SYMBOL_TABLE
"DB_Message"	DB 2	UDT 2
"INS_ZERO_POINT_SYSTEM"	DB 15	FB 15	// Instanzbaustein Nullpunktspannsystem
"INS_CLAMPING_SYSTEM"	DB 17	FB 17	// Instanz-DB Spannsystem (hydraulisch, pneumatisch)
"INS_MESSAGE_OUT"	DB 100	FB 100	// Arbeitsdaten Alarm-/Meldungserfassung
"DB_CK_OP"	DB 101	UDT 101	// DB für Überwachung von Operanden
"DB_IN"	DB 111	DB 111	// Kommunikation - Eingänge
"DB_OUT"	DB 112	DB 112	// Kommunikation - Ausgänge
"ZERO_POINT_SYSTEM"	FB 15	FB 15	// Nullpunktspannsystem
"CLAMPING_SYSTEM"	FB 17	FB 17	// Spannsystem (hydraulisch, pneumatisch)
"AutoSusDoor"	FB 20	FB 20	// pneum.Rüstplatztüren
"MESSAGE_OUT"	FB 100	FB 100	// Ausgabe Alarm-/Betriebsmeldungen
"FlowMonitoring"	FC 10	FC 10	// Strömungsüberwachung
"HydraulicMonitoring"	FC 12	FC 12	// Überwachung Hydrauliksystem (Filter, ...)
"OperatingData"	FC 30	FC 30	// Betriebsdatenerfassung, Signalleuchte (-säule, Ampel)
"MonitoringFuse"	FC 33	FC 33	// Erfassung und Auswertung der Sicherungen
"MontioringCircuitBreaker"	FC 34	FC 34	// Erfassung und Auswertung der Leistungsschalter
"MonitoringMainDrive"	FC 35	FC 35
"ChipConveyor"	FC 42	FC 42
"COOLANT"	FC 50	FC 50	// Kühlmittel Druckerhöhung
"FUNCTIONS"	FC 90	FC 90	// allgemeine Funktionen
"CHANGE_BYTE"	FC 91	FC 91
"SIGNAL"	FC 92	FC 92	// allgemeine Signalverknüpfungen
"SELECT_TIME"	FC 93	FC 93	// aus MD (2Dekaden) 2 Zeitwerte (Time) erzeugen
"MachineType"	FC 94	FC 94	// Dekodierung des Maschinentyps und Optionen aus einem Maschinenparameter
"FC_CK2OP"	FC 101	FC 101	// Überwachung von 2 Operanden
"FC_CK1OP"	FC 102	FC 102	// Überwachung eines Operanden
"INPUT_MASTER"	FC 111	FC 111	// Eingänge von Mastersystem lesen
"OUTPUT_MASTER"	FC 112	FC 112	// Ausgänge an Mastersystem schreiben
"CallAutoSusDoor"	FC 120	FC 120
"INPUT_PERIPHERIE"	FC 121	FC 121	// Eingänge von Peripherie lesen
"OUTPUT_PERIPHERIE"	FC 122	FC 122	// Ausgänge an Peripherie schreiben
"M_LOW"	M 0.0	BOOL	// Merker mit Zustand Low  "FALSE"
"M_HIGH"	M 0.1	BOOL	// Merker mit Zustand High  "TRUE"
"m_expertenbit"	M 0.2	BOOL	// Expertenbit für Fehleranzeige
"M_STARTPULSE"	M 0.5	BOOL	// Startimpuls, wird nur einmalig, für einen Zyklus gesetzt.
"m_inbetriebnahme"	M 0.6	BOOL
"m_konstruktion"	M 0.7	BOOL
"M_TAKT_0.1SEC"	M 1.0	BOOL	// Taktmerker 0.1sec/10Hz
"M_TAKT_0.2SEC"	M 1.1	BOOL	// Taktmerker 0.2sec/5Hz
"M_TAKT_0.4SEC"	M 1.2	BOOL	// Taktmerker 0.4sec/2.5Hz
"M_TAKT_0.5SEC"	M 1.3	BOOL	// Taktmerker 0.5sec/2Hz
"M_TAKT_0.8SEC"	M 1.4	BOOL	// Taktmerker 0.8sec/1.25Hz
"M_TAKT_1.0SEC"	M 1.5	BOOL	// Taktmerker 1.0sec/1Hz
"M_TAKT_1.6SEC"	M 1.6	BOOL	// Taktmerker 1.6sec/0.625Hz
"M_TAKT_2.0SEC"	M 1.7	BOOL	// Taktmerker 2.0sec/0.5Hz
"M_MESSAGE"	M 50.0	BOOL	// Zwischenspeicher für Meldung "PW-Freigabe nicht möglich"
"M_Hyd_Filter_Alarm"	M 50.1	BOOL	// Zwischenspeicher für Hydraulik Filter Alarm
"M_Hyd_Füll_Warn"	M 50.2	BOOL	// Zwischenspeicher für Hydraulik Füllstand Warnung
"M_Hyd_Füll_Alarm"	M 50.3	BOOL	// Zwischenspeicher für Hydraulik Füllstand Alarm
"M_Hyd_Temp_Alarm"	M 50.4	BOOL	// Zwischenspeicher für Hydraulik Temperatur Alarm
"mTypeDMUxxP2"	M 60.1	BOOL	// (1) Maschinenbaureihe DMU xxP2
"mType1"	M 60.2	BOOL
"mType2"	M 60.3	BOOL
"mType3"	M 60.4	BOOL
"mTypeDMCxxU2"	M 60.5	BOOL	// (5) Maschinenbaureihe DMC xxU2
"mTypeDMCxxU2RS"	M 60.6	BOOL	// (6) Maschinenbaureihe DMC xxU2 mit Rundspeicher
"mTypeDMCxxU2WS"	M 60.7	BOOL	// (7) Maschinenbaureihe DMC xxU2 mit Werkstückspeicher (Fastems)
"mType4"	M 61.0	BOOL
"mType5"	M 61.1	BOOL
"mType6"	M 61.2	BOOL
"mType7"	M 61.3	BOOL
"mType8"	M 61.4	BOOL
"mType9"	M 61.5	BOOL
"mType10"	M 61.6	BOOL
"mType11"	M 61.7	BOOL
"mPalletClampingHead"	M 62.0	BOOL	// (256) Palettenausführung mit Spannköpfen/Spannkonen
"mTurnTable"	M 62.1	BOOL	// (512) Fräs-Drehtisch
"mOption2"	M 62.2	BOOL	// (1024)
"mOption3"	M 62.3	BOOL	// (2048)
"mOption4"	M 62.4	BOOL	// (4096)
"mOption5"	M 62.5	BOOL	// (8192)
"mOption6"	M 62.6	BOOL	// (16384)
"mOption7"	M 62.7	BOOL	// (32768)
"mOption8"	M 63.4	BOOL	// (16)
"mOption9"	M 63.5	BOOL	// (32)
"mOption10"	M 63.6	BOOL	// (64)
"mOption11"	M 63.7	BOOL	// (128)
"Flankenmerker_1"	M 80.0	BOOL	// Zwischenspeicher für Flankenauswertung 1
"Flankenmerker_2"	M 80.1	BOOL	// Zwischenspeicher für Flankenauswertung 2
"Flankenmerker_3"	M 80.2	BOOL	// Zwischenspeicher für Flankenauswertung 3
"Flankenmerker_4"	M 80.3	BOOL	// Zwischenspeicher für Flankenauswertung 4
"Flankenmerker_5"	M 80.4	BOOL	// Zwischenspeicher für Flankenauswertung 5
"Flankenmerker_6"	M 80.5	BOOL	// Zwischenspeicher für Flankenauswertung 5
"Flankenmerker_7"	M 80.6	BOOL	// Zwischenspeicher für Flankenauswertung 5
"Flankenmerker_8"	M 80.7	BOOL	// Zwischenspeicher für Flankenauswertung 5
"Hilfsmerker_1"	M 90.0	BOOL	// Zwischenspeicher 1
"Hilfsmerker_2"	M 90.1	BOOL	// Zwischenspeicher 2
"Hilfsmerker_3"	M 90.2	BOOL	// Zwischenspeicher 3
"Hilfsmerker_4"	M 90.3	BOOL	// Zwischenspeicher 4
"Hilfsmerker_5"	M 90.4	BOOL	// Zwischenspeicher 5
"Hilfsmerker_6"	M 90.5	BOOL	// Zwischenspeicher 6
"Hilfsmerker_7"	M 90.6	BOOL	// Zwischenspeicher 7
"Hilfsmerker_8"	M 90.7	BOOL	// Zwischenspeicher 8
"EpxCoolantFlowM7"	M 100.0	BOOL	// Durchflusswächter Kühlmittel2 (M7)
"EpxWireFlowSensorOkM7"	M 100.1	BOOL	// /Durchflusswächter HD Leitungsüberwachung
"EpxCoolantFlowM8"	M 100.2	BOOL	// Durchflusswächter Kühlmittel1 (M8)
"EpxWireFlowSensorOkM8"	M 100.3	BOOL	// /Durchflusswächter ND Leitungsüberwachung
"EPX_ZPS_RELEASE"	M 100.4	BOOL	// Nullpunktspannsystem lösen
"EPX_ZPS_LOCKED"	M 100.5	BOOL	// Nullpunktspannsystem gesperrt
"EPX_ZPS_PRESSURE_MIN1"	M 100.6	BOOL	// Nullpunktspannsystem Drucküberwachung_1 Minimaldruck (p~0) = gespannt
"EPX_ZPS_PRESSURE_MIN2"	M 100.7	BOOL	// Nullpunktspannsystem Drucküberwachung_2 Minimaldruck (p~0) = gespannt
"EPX_ZPS_PRESSURE_MAX1"	M 101.0	BOOL	// Nullpunktspannsystem Drucküberwachung_1 Maximaldruck (p=max) = gelöst
"EPX_ZPS_PRESSURE_MAX2"	M 101.1	BOOL	// Nullpunktspannsystem Drucküberwachung_2 Maximaldruck (p=max) = gelöst
"EPX_COOLANT_LIMIT_VALUE"	M 101.2	BOOL	// /Füllstandsüberwachung im Sammelbehälter
"EPX_LUBRICATION_LEVEL"	M 101.3	BOOL	// Füllstandsüberwachung Schmierstoffaggregat
"EPX_ZPS_MODE_AUTO"	M 101.4	BOOL	// Nullpunktspannsystem in Betriebsart Automatik = Ansteuerung durch ext. Einheit
"EPX_ZPS_INTERLOCK_MIN1"	M 101.5	BOOL	// Nullpunktspannsystem - Verriegelungskontrolle Druck ~0 (drucklos)
"EPX_ZPS_INTERLOCK_MAX1"	M 101.6	BOOL	// Nullpunktspannsystem - Verriegelungskontrolle Druck vorhanden (=verriegelt)
"EPX_ZPS_DISTANCE_P_MIN1"	M 101.7	BOOL	// Nullpunktspannsystem - Auflagenkontrolle Druck ~0 (drucklos)
"EPX_ZPS_DISTANCE_P_MAX1"	M 102.0	BOOL	// Nullpunktspannsystem - Auflagenkontrolle Druck erreicht (Präzision vorhanden)
"EPX_ALARM_QUIT"	M 102.1	BOOL	// Rücksetzen der Fehlermeldung (z.B. Akustik)
"EPX_EL-CABINETDOOR1_OPEN"	M 102.2	BOOL	// Schaltschranktür(-kombination)_1 der Werkzeugmaschine geöffnet
"EPX_EL-CABINETDOOR2_OPEN"	M 102.3	BOOL	// Schaltschranktür(-kombination)_2 der Werkzeugmaschine geöffnet
"EPX_EL-CABINETDOOR5_OPEN"	M 102.4	BOOL	// Schaltschranktür(-kombination)_1 der Kühlschmierstoffanlage geöffnet
"EPX_EL_CABINET_TEMP_1"	M 102.5	BOOL	// Uebertemperatur Schaltschrank Werkzeugmaschine
"EPX_EL_CABINET_TEMP_2"	M 102.6	BOOL	// Grenzwertmeldung Schaltschranktemperatur Werkzeugmaschine
"EPX_EL-CABINETDOOR3_OPEN"	M 102.7	BOOL	// Schaltschranktür(-kombination)_3 der Werkzeugmaschine geöffnet
"EPX_SO_APC_POS_180"	M 103.0	BOOL	// Palettenwechsler Stellung 180 Grad (Palette_2 im Arbeitsraum)
"EPX_SO_APC_POS_0"	M 103.1	BOOL	// Palettenwechsler Stellung 0 Grad (Palette_1 im Arbeitsraum)
"EPX_VCS_MODE_MIXED"	M 103.2	BOOL	// Anwahl Betriebsart <Vakuumsystem Mischbetrieb> aktiv
"EPX_VCS_MODE_VACUUM"	M 103.3	BOOL	// Anwahl Betriebsart <Vakuumsystem Vollwechsel> aktiv
"EPX_VCS_MODE_OFF"	M 103.4	BOOL	// Anwahl Betriebsart <Vakuumsystem Aus>
"EPX_VCS_READY_1"	M 103.5	BOOL	// Betriebsbereitmeldung Vakuumsystem (Arbeitsraum) z.B. Leistungssschalter, ...
"EPX_VCS_READY_2"	M 103.6	BOOL	// Betriebsbereitmeldung Vakuumsystem (Rüstplatz) z.B. Leistungssschalter, ...
"EPX_VCS_RELEASE_FIXTURE2"	M 103.7	BOOL	// Vakuumspannsystem am Rüstplatz lösen
"EPX_VCS_FIXTURE1_1_P=0"	M 104.0	BOOL	// Vakuumspannsystem im Arbeitsraum Drucklos (=gelöst)
"EPX_VCS_FIXTURE1_2_P=0"	M 104.1	BOOL	// Vakuumspannsystem im Arbeitsraum Drucklos (=gelöst)
"EPX_VCS_FIXTURE2_1_P=0"	M 104.2	BOOL	// Vakuumspannsystem am Rüstplatz Drucklos (=gelöst)
"EPX_VCS_FIXTURE1_1_P=MAX"	M 104.3	BOOL	// Vakuumspannsystem im Arbeitsraum gespannt (eingestellter Sollwert erreicht)
"EPX_VCS_FIXTURE2_1_P=MAX"	M 104.4	BOOL	// Vakuumspannsystem am Rüstplatz gespannt (eingestellter Sollwert erreicht)
"EpxHydrFilterAlarm1NC"	M 104.5	BOOL	// Filterverschmutzung Hydraulikfilter-Maschine (Alarm 100%)
"EpxHydrFilterWarning1NC"	M 104.6	BOOL	// Filterverschmutzung Hydraulikfilter-Maschine (Warnung 75%)
"EPX_EXH_NEG_READY1"	M 104.7	BOOL	// Auswertung Leistungsschalter des Nebelabscheiders_1/Absaugung_1
"EPX_EXH_ON1"	M 105.0	BOOL	// Überwachung Ansteuerung Nebelabscheider_1, Gerät ein
"EPX_MACHINE_ON_K1"	M 105.1	BOOL	// "Maschine Ein"-Signal an Kühlschmierstoffanlage (kein Not-Aus)
"EPX_WORKROOM_CLOSED_K1"	M 105.2	BOOL	// "Arbeitsraumtüren geschlossen"-Signal an Kühlschmierstoffanlage
"EPX_NEG_COO_MESSAGE"	M 105.3	BOOL	// Warnmeldung von Kühlschmierstoffanlage
"EPX_NEG_COO_ALARM"	M 105.4	BOOL	// Störung, Alarm von Kühlschmierstoffanlage
"EPX_COO_ACK_COOLANT2.2"	M 105.5	BOOL	// Rückmeldung wenn Druckstufe_2 von Kühlmittel_2 erreicht wurde (YD-Anlauf)
"EPX_COO_MAINVALVE_CLOSED"	M 105.6	BOOL	// Kühlschmierstoffzufuhr Haupt-/Zentralventil geschlossen
"EPX_COO_PRESSURE_P=MAX"	M 105.7	BOOL	// Kühlschmierstoffzufuhr Drucküberwachung
"EPX_COO_MAIN_FLOW"	M 106.0	BOOL	// Kühlschmierstoffzufuhr Durchflussüberwachung
"EPX_COO_LIMITVALUE_K5"	M 106.1	BOOL	// Grenzwertmeldung aus Sammelbehälter (SPF) z.B. von WHG-Sonde
"EPX_NEG_COO_FILTALARM2.2"	M 106.2	BOOL	// Filterverschmutzung Feinfilter Alarmmeldung für KSS-Zufuhr_2 (IKZ)-Druckstufe_2
"EPX_COO_FILTWARN2.2"	M 106.3	BOOL	// Filterverschmutzung Feinfilter Warnmeldung für KSS-Zufuhr_2 (IKZ) - Druckstufe_2
"EPX_VCS_RELEASE_FIXTURE1"	M 106.4	BOOL	// Vakuumspannsystem im Arbeitsraum lösen
"EPX_CS_OFF"	M 106.5	BOOL	// Spannsystem deaktiviert, Aus
"EPX_CS_MODE_AUTO"	M 106.6	BOOL	// Spannsystem in der Betriebsart "AUTOMATIK" (=externe Ansteuerung)
"EPX_CS_RELEASE1_1"	M 106.7	BOOL	// Anforderung Spannsystem lösen im Arbeitsraum (Spannkreis 1)
"EPX_CS_PRESSURE1_1MIN"	M 107.0	BOOL	// Spannsystem DruckÜW im Arbeitsraum (Spannkreis 1/Stufe 1 - Systemdruck Min)
"EPX_CS_PRESSURE1_1MAX"	M 107.1	BOOL	// Spannsystem DruckÜW im Arbeitsraum (Spannkreis 1/Stufe 1 - Systemdruck Max)
"EPX_CS_PRESSURE1_2MIN"	M 107.2	BOOL	// Spannsystem DruckÜW im Arbeitsraum (Spannkreis 1/Stufe 2 - Lösedruck Min)
"EPX_CS_PRESSURE1_2MAX"	M 107.3	BOOL	// Spannsystem DruckÜW im Arbeitsraum (Spannkreis 1/Stufe 2 - Lösedruck Max)
"EPX_CS_STROKE1_POS1"	M 107.4	BOOL	// Spannsystem Hubkontrolle im Arbeitsraum (Werkstück gelöst)
"EPX_CS_STROKE1_POS2"	M 107.5	BOOL	// Spannsystem Hubkontrolle im Arbeitsraum (Werkstück gespannt)
"EPX_CS_STROKE1_POS3"	M 107.6	BOOL	// Spannsystem Hubkontrolle im Arbeitsraum (gespannt ohne Werkstück)
"EPX_EXT_FIXTURE_EXIST"	M 107.7	BOOL	// Werkstück an Spannvorrichtung, Spannfutter (Signal von externer Einheit)
"EPX_EXT_RELEASE1"	M 108.0	BOOL	// Anforderung Spannsystem lösen im Arbeitsraum (Signal von externer Einheit)
"EPX_APC_DOOR_CLOSED"	M 108.1	BOOL	// Rüstplatztüren geschlossen (NICHT verriegelt)
"EPX_EXH_ON2"	M 108.2	BOOL	// Überwachung Ansteuerung Nebelabscheider_2, Gerät ein
"EPX_EXH_NEG_READY2"	M 108.3	BOOL	// Auswertung Leistungsschalter des Nebelabscheiders_2/Absaugung_2
"EPX_EXH_SELECT1"	M 108.4	BOOL	// Absaugung - Auswahl für Nebelabscheider_1
"EPX_EXH_SELECT2"	M 108.5	BOOL	// Absaugung - Auswahl für Nebelabscheider_2
"EPX_MCS_CLAMP1"	M 108.6	BOOL	// Magnetspannsystem_1 spannen
"EPX_MCS_RELEASE1"	M 108.7	BOOL	// Magnetspannsystem_1 lösen
"EPX_MCS_PARK_STATION1"	M 109.0	BOOL	// Magnetspannsystem_1 Magnetisierungsstecker am Ablageplatz (Parkstation)-Rpl
"EPX_MCS_LOCKED1"	M 109.1	BOOL	// Magnetspannsystem_1 Betriebsart gesperrt/deaktiviert
"EPX_HYD_FILTER_OK1"	M 109.2	BOOL	// Filter des Hydraulikaggregates-Maschine in Ordnung
"EPX_COO_ACK_COOLANT2.1"	M 109.3	BOOL	// Rückmeldung wenn Druckstufe_1 von Kühlmittel_2 erreicht wurde (YD-Anlauf)
"EPX_ZPS_RELEASE1_START"	M 109.4	BOOL	// Nullpunktspannsystem lösen - Startsignal, direkt vom Befehlsgerät
"EPX_SRT_SWIVELPOS=0"	M 109.5	BOOL	// Schwenkrundtisch - Schwenkachse steht in horizontaler Position (0 Grad)
"EPX_CS_FINALPOS0"	M 109.6	BOOL	// Spannvorrichtung - Endlage Position 0 erreicht
"EPX_CS_FINALPOS1"	M 109.7	BOOL	// Spannvorrichtung - Endlage Position 1 erreicht
"EPX_CS_NOT_FINALPOS0"	M 110.0	BOOL	// Spannvorrichtung - Endlage Position 0  NICHT erreicht/vorhanden
"EPX_CS_NOT_FINALPOS1"	M 110.1	BOOL	// Spannvorrichtung - Endlage Position 1  NICHT erreicht/vorhanden
"EPX_CS_PRESSURIZED_POS0"	M 110.2	BOOL	// Spannvorrichtung - Druck vorhanden für Bewegung auf Position 0
"EPX_CS_PRESSURIZED_POS1"	M 110.3	BOOL	// Spannvorrichtung - Druck vorhanden für Bewegung auf Position 1
"EPX_CS_ROTATECONTROL_ON"	M 110.4	BOOL	// Spannvorrichtung - Überwachung der Drehbewegung aktiviert
"EPX_COO_FLUSH1_P=SYST"	M 110.5	BOOL	// Drucküberwachung Kühlschmierstoffzufuhr Spänespülung(en) = Systemdruck
"EPX_COO_FLUSH1_P=MAX"	M 110.6	BOOL	// Drucküberwachung Kühlschmierstoffzufuhr Spänespülung(en) = maximaler Druck
"EPX_ZPS_ENABLE"	M 110.7	BOOL	// Nullpunktspannsystem gespannt oder nicht aktiviert (?HLS?)
"EPX_MMS_FILLUNIT_NIV_MIN"	M 111.0	BOOL	// MMS: Versorgungseinheit - Füllstand Minimum
"EPX_MMS_NIVEAU_MIN"	M 111.1	BOOL	// MMS: Füllstand Minimum
"EPX_MMS_NIVEAU_MAX"	M 111.2	BOOL	// MMS: Füllstand Maximum
"EPX_MMS_NIVEAU_WAR_MIN"	M 111.3	BOOL	// MMS: Füllstand Minimum - Vorwarnung
"EPX_SPINDLE_FEED_STOP"	M 111.4	BOOL	// Spindel- und Vorschub Halt (allgemein)
"EPX_VCS_FIXTURE_START1"	M 111.5	BOOL	// Vakuumsystem lösen (Startsignal)
"EPX_MCS_MODE_ON1"	M 111.6	BOOL	// Magnetspannsystem (Hauptschalter Ein)
"EPX_ZPS_CYL_LIFT"	M 111.7	BOOL	// Nullpunktspannsystem Abhebezylinder heben (ausfahren)
"EPX_ZPS_CYL_LOWER"	M 112.0	BOOL	// Nullpunktspannsystem Abhebezylinder senken (einfahren)
"EPX_ZPS_CYL_PRESS_MIN1"	M 112.1	BOOL	// Nullpunktspannsystem Abhebezylinder Heben Druck Minimum   (p~0) = eingefahren
"EPX_ZPS_CYL_PRESS_MIN2"	M 112.2	BOOL	// Nullpunktspannsystem Abhebezylinder Senken Druck Minimum   (p~0) = ausgefahren
"EPX_ZPS_CYL_PRESS_MAX1"	M 112.3	BOOL	// Nullpunktspannsystem Abhebezylinder Heben Druck Maximum   (p~max) = ausgefahren
"EPX_ZPS_CYL_PRESS_MAX2"	M 112.4	BOOL	// Nullpunktspannsystem Abhebezylinder Senken Druck Maximum   (p~max) = eingefahren
"EpxFunctionM86"	M 112.5	BOOL	// maschinenspezifische Funktion (M86)
"EpxFunctionM87"	M 112.6	BOOL	// maschinenspezifische Funktion (M87)
"EpxFunctionM88"	M 112.7	BOOL	// maschinenspezifische Funktion (M88)
"EpxFunctionM89"	M 113.0	BOOL	// maschinenspezifische Funktion (M89)
"EpxMcsParkshutterLocked"	M 113.1	BOOL	// Magnetspannsystem Parkstation Klappe geschlossen
"EpxMcsAntiSteckParks"	M 113.2	BOOL	// Magnetspannsystem Stecker nicht vorhanden
"EpxMcsParkstatEnable"	M 113.3	BOOL	// Magnetspannsystem Parkstation entriegelt
"EpxMcsPlugIn"	M 113.4	BOOL	// Magnetspannsystem Stecker in Magnetspannplatte
"EpxMcsOff"	M 113.5	BOOL	// Magnetspannsystem aus
"EpxMcsEnableRelease"	M 113.6	BOOL	// Magnetspannsystem Freigabe lösen
"EpxMcsMaleInParkstaion"	M 113.7	BOOL	// Magnetspannsystem Stecker in Parkstation
"EpxMcsAdhesivForceOk"	M 114.0	BOOL	// Magnetspannsystem eingestellte Haftkraftstufe erreicht
"EpxCooPwarnSupfineLevel"	M 114.1	BOOL	// Vorwarnung Füllstand Kühlschmierstoff im Feinbereich
"EpxCooEnergyCentrifugeOk"	M 114.2	BOOL	// Überwachung Leistungsschalter der Zentrifuge
"EpxCooCentrifugeReady"	M 114.3	BOOL	// Zentrifuge Betreibsbereit
"EpxCooCentrifugeRun"	M 114.4	BOOL	// Zentrifuge in Betrieb
"EpxCooPwarnCentrifugeQui"	M 114.5	BOOL	// Vorwarnung der Zentrifuge zurücksetzen
"EPX_ZPS_CS1_PRESSLES"	M 114.6	BOOL	// Abfrage des Spanndruckes der Spannhydraulik Kreis 1
"EPX_ZPS_CS2_PRESSLES"	M 114.7	BOOL	// Abfrage des Spanndruckes der Spannhydraulik Kreis 2
"EpxExhausterModeAuto"	M 115.0	BOOL	// Automatikbetrieb Absaugung Ölnebelabscheider
"EPX_SAMMELSTÖRUNG_1"	M 115.1	BOOL	// Meldung von externer Meldeeinrichtung
"EPX_SAMMELSTÖRUNG_2"	M 115.2	BOOL	// Meldung von externer Meldeeinrichtung
"EpxCooNoLimitCollBasin"	M 115.3	BOOL	// keine Grenzwertmeldung Sammelbehälter (WHG)
"EpxEmergStopMachineNC"	M 115.4	BOOL	// Kein Not-Aus an Werkzeugmaschine betätigt
"EpxEmergStopPanel"	M 115.5	BOOL	// Not-Aus Pilzdrucktaster an Bedienpult (Werkzeugmaschine) betätigt
"EpxEmergStopChipConv"	M 115.6	BOOL	// Not-Aus Pilzdrucktaster am Späneförderer betätigt
"EpxEmergStopSetUpStat"	M 115.7	BOOL	// Not-Aus Pilzdrucktaster am Rüstplatz (Palettenspeicher) betätigt
"EpxEmergStopToolInpStat"	M 116.0	BOOL	// Not-Aus Pilzdrucktaster an der Werkzeugeingabestation betätigt
"EpxLubricatPressureXaxis"	M 116.1	BOOL	// Drucküberwachung Schmierung Verteiler X-Achse Ok
"EpxLubricatPressureYaxis"	M 116.2	BOOL	// Drucküberwachung Schmierung Verteiler Y-Achse Ok
"EpxLubricatPressureZaxis"	M 116.3	BOOL	// Drucküberwachung Schmierung Verteiler Z-Achse Ok
"EpxFaultExtChipConveyNC"	M 116.4	BOOL	// LOW = Störung an externem (zentralen) Späneförderer
"EpxLimitValveCoolantNC"	M 116.5	BOOL	// LOW = maximaler Füllstand (Grenzwert) der Kühlschmierstoffanlage erreicht/übers.
"EpxMaintDoorToolInpStat"	M 116.6	BOOL	// Wartungstüre Werkzeugeingabestation offen
"EpxMaintDoorToolMag"	M 116.7	BOOL	// Wartungstüre Werkzeugmagazin offen
"EpxMaintDoorPalletStor"	M 117.0	BOOL	// Wartungstüre Palettenspeicher/-wechsler offen
"EpxLubTablePreExi"	M 117.1	BOOL	// NC-Rundtisch Schmierung Druck Vorhanden
"EpxEmergStopHaWhToolMag"	M 117.2	BOOL	// Not-Aus Pilzdrucktaster des Handrad vom Werkzeugmagazin betätigt
"EpxLubTableApsOk"	M 117.3	BOOL	// Schmierstoffpumpe Leistungsschalter Ok
"EpxLubXAxisPreExi1"	M 117.4	BOOL	// Drucküberwachung Schmierung Verteiler KUG X-Achse
"EpxLubYAxisPreExi1"	M 117.5	BOOL	// Drucküberwachung Schmierung Verteiler KUG Y-Achse
"EpxLubPcAxisPreExi"	M 117.6	BOOL	// Drucküberwachung Schmierung Verteiler Palettenspeichersystem (Palettenwechsler)
"EpxLubSstAxisPreExi"	M 117.7	BOOL	// Drucküberwachung Schmierung Verteiler Ruestplatz
"EpxFusePlugIndicPlate"	M 118.0	BOOL	// Überwachung Sicherungsautomat Steckdose Frontschild
"EpxFuseLubPump"	M 118.1	BOOL	// Überwachung Sicherungsautomat Schmierstoffpumpe
"EpxFuseAsi"	M 118.2	BOOL	// Überwachung Sicherungsautomat AS-i Netzteil
"EpxFuseFlowControl"	M 118.3	BOOL	// Überwachung Sicherungsautomat Durchflusswächter
"EpxFuseLightBulbs"	M 118.4	BOOL	// Überwachung Sicherungsautomat Leuchtmelder Kommandostation
"EpxFuseControlCircuit"	M 118.5	BOOL	// Überwachung Sicherungsautomat Steuerstromkreis
"EpxFuseCncControl"	M 118.6	BOOL	// Überwachung Sicherungsautomat CNC-Steuerung
"EpxFuseEmpStopConCircuit"	M 118.7	BOOL	// Überwachung Sicherungsautomat NOT-AUS Steuerstromkreis
"EpxFuseToolChanger"	M 119.0	BOOL	// Überwachung Sicherungsautomat Werkzeugwechsler
"EpxFuseDcControlVoltage"	M 119.1	BOOL	// Überwachung Sicherungsautomat DC-Steuerspannung
"EpxFusePalletChanger"	M 119.2	BOOL	// Überwachung Sicherungsautomat Palettenwechsler
"EpxFuseCoolantUnit"	M 119.3	BOOL	// Überwachung Sicherungsautomat Kühlmittelanlage
"EpxFusePcu50"	M 119.4	BOOL	// Überwachung Sicherungsautomat PCU 50
"EpxFuseScreen"	M 119.5	BOOL	// Überwachung Sicherungsautomat Bildschirm
"EpxFuseMachineIm151_4"	M 119.6	BOOL	// Überwachung Sicherungsautomat Maschine IM 151
"EpxFuseMachineOutp1Im151"	M 119.7	BOOL	// Überwachung Sicherungsautomat Ausgänge Maschine IM 151
"EpxFuseMachineOutp2Im151"	M 120.0	BOOL	// Überwachung Sicherungsautomat Ausgänge Maschine IM 151
"EpxFuseSpeedControl"	M 120.1	BOOL	// Überwachung Sicherungsautomat Drehzahl Überwachung
"EpxFusePowerPacTc"	M 120.2	BOOL	// Überwachung Sicherungsautomat Netzteil Werkzeugwechsler
"EpxFuseToolIdentificatio"	M 120.3	BOOL	// Überwachung Sicherungsautomat Werkzeugidentifikation
"EpxFuseToolCone"	M 120.4	BOOL	// Überwachung Sicherungsautomat Werkzeugkegel
"EpxFuseControCirPis"	M 120.5	BOOL	// Überwachung Sicherungsautomat Palettenspeichersystem
"EpxFuseBrakePs"	M 120.6	BOOL	// Überwachung Sicherungsautomat Palettenspeichersystem Bremse
"EpxFuseOperaDataRecord"	M 120.7	BOOL	// Überwachung Sicherungsautomat Betriebsdatenerfassung
"EpxFuseToolBrake"	M 121.0	BOOL	// Überwachung Sicherungsautomat Werkzeugbruchüberwachung
"EpxFuseMms"	M 121.1	BOOL	// Überwachung Sicherungsautomat Minimalmengenschmierung
"EpxFuseSlave8"	M 121.2	BOOL	// Überwachung Sicherungsautomat Tuning IM 151
"EpxFuseSlave8Output"	M 121.3	BOOL	// Überwachung Sicherungsautomat Tuning Ausgänge IM 151
"EpxFuseSlave8Input"	M 121.4	BOOL	// Überwachung Sicherungsautomat Tuning Eingänge IM 151
"EpxFuseCabinetLightning"	M 121.5	BOOL	// Überwachung Sicherungsautomat Schaltschrankbeleuchtung
"EpxCuFuseSensor"	M 121.6	BOOL	// Überwachung Sicherungsautomat Sensoren Kühlmittelanlage
"EpxCuFusePropValve1"	M 121.7	BOOL	// Überwachung Sicherungsautomat Proportionalventil 1 Kühlmittelanlage
"EpxCuFusePropValve2"	M 122.0	BOOL	// Überwachung Sicherungsautomat Proportionalventil 2 Kühlmittelanlage
"EpxCuApsCoolant1"	M 122.1	BOOL	// Überwachung Leistungsschalter Kühlmittel 1
"EpxCuApsFlushCleaTop"	M 122.2	BOOL	// Überwachung Leistungsschalter Spänespülung Dach
"EpxCuApsFlushGun"	M 122.3	BOOL	// Überwachung Leistungsschalter Spülpistole
"EpxCuApsFlushCleaCabDoor"	M 122.4	BOOL	// Überwachung Leistungsschalter Spänespülung Kabinentür
"EpxCuApsSuperfineRegion"	M 122.5	BOOL	// Überwachung Leistungsschalter Feinstbereich
"EpxCuApsTroughScraper"	M 122.6	BOOL	// Überwachung Leistungsschalter Kratzerförderer
"EpxCuMainSwitch"	M 122.7	BOOL	// Überwachung Hauptschalter Kühlmittelanlage
"EpxCuApsPump40bar"	M 123.0	BOOL	// Überwachung Leistungsschalter Hochdruckpumpe 40 bar
"EpxCuApsPump80bar"	M 123.1	BOOL	// Überwachung Leistungsschalter Hochdruckpumpe 80 bar
"EpxCuTempApsCompressor"	M 123.2	BOOL	// Überwachung Leistungsschalter Kompressor Kühlaggregat
"EpxCuTempApsFan"	M 123.3	BOOL	// Überwachung Leistungsschalter Lüfter Kühlaggregat
"EpxCuTempApsAgitator"	M 123.4	BOOL	// Überwachung Leistungsschalter Rührwerk Kühlaggregat
"EpxCuTempApsLiftingPump"	M 123.5	BOOL	// Überwachung Leistungsschalter Hebepumpe Kühlaggregat
"EpxCuTempApsHeating"	M 123.6	BOOL	// Überwachung Leistungsschalter Heizung Kühlaggregat
"EpxCuTempApsContrVoltage"	M 123.7	BOOL	// Überwachung Leistungsschalter Steuerspannung Kühlaggregat
"EpxApsCabinetLightning"	M 124.0	BOOL	// Überwachung Leistungsschalter Schaltschrankbeleuchtung
"EpxApsDcControlVoltage1"	M 124.1	BOOL	// Überwachung Leistungsschalter DC-Steuerspannung 1
"EpxApsDcControlVoltage2"	M 124.2	BOOL	// Überwachung Leistungsschalter DC-Steuerspannung 2
"EpxApsAcControlVoltage"	M 124.3	BOOL	// Überwachung Leistungsschalter AC-Steuerspannung
"EpxApsTemperature"	M 124.4	BOOL	// Überwachung Leistungsschalter Kuehl/Heizaggregat
"EpxApsPowerSupplyModule"	M 124.5	BOOL	// Überwachung Leistungsschalter AC-Versorgungsmodul
"EpxMcsParkStation2"	M 124.6	BOOL	// Magnetspannsystem_2 Magnetisierungsstecker am Ablageplatz (Parkstation)-Maschine
"EpxMcsReleased"	M 124.7	BOOL	// Magnetspannplatte gelöst
"EpxMcsChucked"	M 125.0	BOOL	// Magnetspannplatte gespannt
"EpxMcsMalfunction"	M 125.1	BOOL	// Magnetspannsystem Störung
"EpxFeedStop"	M 125.2	BOOL	// Vorschub Halt
"EpxFuseMachineIm151_7"	M 125.3	BOOL	// Überwachung Sicherungsautomat Maschine IM 151_7
"EpxFuseSpeedControlSst"	M 125.4	BOOL	// Überwachung Sicherungsautomat Drehzahl Überwachung Rüstplatz
"EpxFuseMeasuringSensor"	M 125.5	BOOL	// Überwachung Sicherungsautomat Messtaster
"EpxFuseWorkingAreaDoor"	M 125.6	BOOL	// Überwachung Sicherungsautomat Kabinentüre
"EpxTmsFuseBrake"	M 125.7	BOOL	// Überwachung Sicherungsautomat Bremse Regalmagazin
"EpxTmsFuseAcContrVoltage"	M 126.0	BOOL	// Überwachung Sicherungsautomat AC-Steuerspannung Regalmagazin
"EpxTmsFuseControlCircuit"	M 126.1	BOOL	// Überwachung Sicherungsautomat Steuerstromkreis Regalmagazin
"EpxTmsFuseControlPanel"	M 126.2	BOOL	// Überwachung Sicherungsautomat Werkzeugeingabestation Regalmagazin
"EpxTmsFuseOutput"	M 126.3	BOOL	// Überwachung Sicherungsautomat Ausgänge Regalmagazin
"EpxTmsFusePowerPac"	M 126.4	BOOL	// Überwachung Sicherungsautomat Netzteil Regalmagazin
"EpxTmsApsPower"	M 126.5	BOOL	// Überwachung Leistungschalter Netzeinspeisung Regalmagazin
"EpxLubTmsAxisPreExi"	M 126.6	BOOL	// Drucküberwachung Schmierung Verteiler Werkzeugmagazin
"EpxFuseFeedDrive"	M 126.7	BOOL	// Überwachund Sicherungsautomat Leistung Spindel
"EpxMaintDoorToolShelf"	M 127.0	BOOL	// Wartungstüre Werkzeugregal offen
"EpxApsAcControVoltageFan"	M 127.1	BOOL	// Überwachung Leistungsschalter Lüfter AC
"EpxApsAcCoolCabinet"	M 127.2	BOOL	// Überwachung Leistungsschalter Kühlaggregat Schaltschrank
"EpxApsPowerToolShelf"	M 127.3	BOOL	// Überwachung Leistungsschalter Werkzeugregal
"EpxApsFdFan"	M 127.4	BOOL	// Überwachung Leistungsschalter Lüfter FD
"EpsApsCoolingUnit"	M 127.5	BOOL	// Überwachung Leistungsschalter Kühlmittelanlage
"EpxTmsApsAcControlVoltag"	M 127.6	BOOL	// Überwachung Leistungsschalter Steuerspannung AC-Regalmagazin
"EpxTmsApsDrives"	M 127.7	BOOL	// Überwachung Leistungsschalter Antriebe Regalmagazin
"EpxHydFuellMaxOk"	M 128.0	BOOL	// Füllstand Hydraulik Maximum Ok
"EpxHydFuellMinOk"	M 128.1	BOOL	// Füllstand Hydraulik Minimum Ok
"EpxFuse230V"	M 128.2	BOOL	// Überwachung Sicherungsautomaten 230V
"EpxFuse24V"	M 128.3	BOOL	// Überwachung Sicherungsautomaten 24V
"EpxApsContPanelPlugSock"	M 128.4	BOOL	// Überwachung Leistungsschalter Steckdose Bedienpult
"EpxApsPcPlugSock"	M 128.5	BOOL	// Überwachung Leistungsschalter Steckdose Palettenwechsler-/speichersystem
"EpxSusDoorSystPressMax"	M 128.6	BOOL	// Ruestplatztürantreib Systemdruck vorhanden
"EpxCloseSusDoor"	M 128.7	BOOL	// Rüstplatztüre(n) schliessen (manuelle Bedienung)
"EpxOpenSusDoor"	M 129.0	BOOL	// Rüstplatztüre(n) öffnen (manuelle Bedienung)
"EpxRobotLock"	M 129.1	BOOL	// Betreibsart Werkstücklader gesperrt = manuelles Beladen
"EpxSafetyEdgeSusDoor"	M 129.2	BOOL	// Schaltleiste an Rüstplatztüren betätigt
"EpxSusDoorPressMonOpen"	M 129.3	BOOL	// Drucküberwachung Rüstplatztüren öffnen aktiv
"EpxSusDoorPressMonClose"	M 129.4	BOOL	// Drucküberwachung Rüstplatztüren schließen aktiv
"EpxSusDoorLeftOpen"	M 129.5	BOOL	// Rüstplatztüre links vollständig geöffnet
"EpxSusDoorRightOpen"	M 129.6	BOOL	// Rüstplatztüre rechts vollständig geöffnet
"EpxSusDoorClosed"	M 129.7	BOOL	// Rüstplatztüre(n) geschlossen
"EpxSusDoorClosedLocked"	M 130.0	BOOL	// Rüstplatztüre(n) geschlossen und verriegelt
"EpxPressMonitLubToolMag"	M 130.1	BOOL	// Drucküberwachung Schmierung Werkzeugmagazin
"EpxCircBrkMachineOutpNc"	M 130.2	BOOL	// Überwachung Leitungsschutzschalter Ausgänge IM151 (Maschine)
"EpxCircBrkCtlVoToolMagNc"	M 130.3	BOOL	// Überwachung Leitungsschutzschalter Steuerstromkreis Werkzeugmagazin
"EpxPowSwitchAddCoolng1Nc"	M 130.4	BOOL	// Überwachung Leitungsschutzschalter Kühlaggregat Zusatzschaltschrank (Einspeisung
"EpxApsWorkingAreaDoor"	M 130.5	BOOL	// Überwachung Leistungschutzschalter Kabinentüre
"EpxMachineOn"	M 130.6	BOOL	// Maschine ist eingeschaltet (kein Not-Aus)
"EpxProgramRun"	M 130.7	BOOL	// Programm läuft
"EpxLubDec1Bit_0"	M 131.0	BOOL	// Schmierimpuls Binär codiert Bit 0
"EpxLubDec1Bit_1"	M 131.1	BOOL	// Schmierimpuls Binär codiert Bit 1
"EpxLubDec1Bit_2"	M 131.2	BOOL	// Schmierimpuls Binär codiert Bit 2
"EpxLubDec1Bit_3"	M 131.3	BOOL	// Schmierimpuls Binär codiert Bit 3
"EpxLubDec1Bit_4"	M 131.4	BOOL	// Schmierimpuls Binär codiert Bit 4
"EpxLubDec1Bit_5"	M 131.5	BOOL	// Schmierimpuls Binär codiert Bit 5
"EpxLubDec1Bit_6"	M 131.6	BOOL	// Schmierimpuls Binär codiert Bit 6
"EpxLubDec1Bit_7"	M 131.7	BOOL	// Schmierimpuls Binär codiert Bit 7
"EpxLubDec2Bit_0"	M 132.0	BOOL	// Pausenzeit Binär codiert Bit 0
"EpxLubDec2Bit_1"	M 132.1	BOOL	// Pausenzeit Binär codiert Bit 1
"EpxLubDec2Bit_2"	M 132.2	BOOL	// Pausenzeit Binär codiert Bit 2
"EpxLubDec2Bit_3"	M 132.3	BOOL	// Pausenzeit Binär codiert Bit 3
"EpxLubDec2Bit_4"	M 132.4	BOOL	// Pausenzeit Binär codiert Bit 4
"EpxLubDec2Bit_5"	M 132.5	BOOL	// Pausenzeit Binär codiert Bit 5
"EpxLubDec2Bit_6"	M 132.6	BOOL	// Pausenzeit Binär codiert Bit 6
"EpxLubDec2Bit_7"	M 132.7	BOOL	// Pausenzeit Binär codiert Bit 7
"IpxAxisStop"	M 133.0	BOOL	// Stillstand der Achsen
"EpxRoutingBit1"	M 133.1	BOOL	// Datensignal von digitalem Eingang<IX_ROUTING_BIT_0
"EpxRoutingBit2"	M 133.2	BOOL	// Datensignal von digitalem Eingang<IX_ROUTING_BIT_0
"EpxRoutingBit3"	M 133.3	BOOL	// Datensignal von digitalem Eingang<IX_ROUTING_BIT_0
"EpxRoutingBit4"	M 133.4	BOOL	// Datensignal von digitalem Eingang<IX_ROUTING_BIT_0
"EpxRoutingBit5"	M 133.5	BOOL	// Datensignal von digitalem Eingang<IX_ROUTING_BIT_0
"EpxRoutingBit6"	M 133.6	BOOL	// Datensignal von digitalem Eingang<IX_ROUTING_BIT_0
"EpxRoutingBit7"	M 133.7	BOOL	// Datensignal von digitalem Eingang<IX_ROUTING_BIT_0
"EpxRoutingBit8"	M 134.0	BOOL	// Datensignal von digitalem Eingang<IX_ROUTING_BIT_0
"EpxRoutingBit9"	M 134.1	BOOL	// Datensignal von digitalem Eingang<IX_ROUTING_BIT_0
"EpxRoutingBit10"	M 134.2	BOOL	// Datensignal von digitalem Eingang<IX_ROUTING_BIT_0
"EpxRoutingBit11"	M 134.3	BOOL	// Datensignal von digitalem Eingang<IX_ROUTING_BIT_0
"EpxRoutingBit12"	M 134.4	BOOL	// Datensignal von digitalem Eingang<IX_ROUTING_BIT_0
"EpxRoutingBit13"	M 134.5	BOOL	// Datensignal von digitalem Eingang<IX_ROUTING_BIT_0
"EpxRoutingBit14"	M 134.6	BOOL	// Datensignal von digitalem Eingang<IX_ROUTING_BIT_0
"EpxRoutingBit15"	M 134.7	BOOL	// Datensignal von digitalem Eingang<IX_ROUTING_BIT_0
"EpxCooHighPressure_P=Max"	M 135.0	BOOL	// Kühlschmierstoffzufuhr Drucküberwachung Hochdruckkreis
"EpxCooLowPressure_P=Max"	M 135.1	BOOL	// Kühlschmierstoffzufuhr Drucküberwachung Niederdruckkreis
"EpxCooMainValveHpClosed"	M 135.2	BOOL	// Kühlschmierstoffzufuhr Hauptventil Hochdruck geschlossen
"EpxCooMainValveLpClosed"	M 135.3	BOOL	// Kühlschmierstoffzufuhr Hauptventil Niederdruck geschlossen
"EpxCcCountclockwise_2"	M 135.4	BOOL	// Ansteuerung Zusatzspäneförderer Linkslauf
"EpxCcClockwise_2"	M 135.5	BOOL	// Ansteuerung Zusatzspäneförderer Rechtslauf
"EpxCcAutomatic_2"	M 135.6	BOOL	// Ansteuerung Zusatzspäneförderer Automatikbetrieb
"EpxCcManuel_2"	M 135.7	BOOL	// Ansteuerung Zusatzspäneförderer Handbetrieb
"EpxHydTemperatureMonitor"	M 136.0	BOOL	// Temperatureüberwachung des Hydraulikaggregats Maschine
"EpxFunktionM80"	M 136.1	BOOL	// maschinenspezifische Funktion (M80)
"EpxFunktionM81"	M 136.2	BOOL	// maschinenspezifische Funktion (M81)
"EpxFunktionM82"	M 136.3	BOOL	// maschinenspezifische Funktion (M82)
"EpxFunktionM83"	M 136.4	BOOL	// maschinenspezifische Funktion (M83)
"EpxFunktionM84"	M 136.5	BOOL	// maschinenspezifische Funktion (M84)
"EpxFunktionM85"	M 136.6	BOOL	// maschinenspezifische Funktion (M85)
"EpxGenMTHFeedback"	M 136.7	BOOL	// Rückmeldung M-Funktion
"EpxCsHydrFilterWarn1NC"	M 137.0	BOOL	// Filterverschmutzung Hydraulikfilter-Spannhydraulik Maschine (Warnung) 75%
"EpxCsHydrFilterAlarm1NC"	M 137.1	BOOL	// Filterverschmutzung Hydraulikfilter-Spannhydraulik Maschine (Alarm) 100%
"IpxCooPneumSystPressMax"	M 137.2	BOOL	// Überwachung Pneumatikdruck vorhanden (KSS-Versorgung)
"ApxStatusLightGreen"	M 180.0	BOOL	// Signalleuchte (Ampel) Element: GRÜN (GN)
"ApxStatusLightYellow"	M 180.1	BOOL	// Signalleuchte (Ampel) Element: GELB (YE)
"ApxStatusLightRed"	M 180.2	BOOL	// Signalleuchte (Ampel) Element: ROT (RD)
"APX_BDE_AXIS_SPINDLE"	M 180.3	BOOL	// mindestens 1Achse und Spindel aktiv
"APX_BDE_MACHINE_ON"	M 180.4	BOOL	// Maschine Ein (kein Not-Aus)
"APX_MODE_MANUAL"	M 180.5	BOOL	// Betriebsart "MANUAL"
"APX_MODE_TEACH_IN"	M 180.6	BOOL	// Betriebsart "TEACH IN"
"APX_MODE_AUTOMATIK"	M 180.7	BOOL	// Betriebsart "AUTOMATIK"
"ApxFeedOverride>x%"	M 181.0	BOOL	// Vorschubpotentiometer größer Wert "X"
"APX_CNC_ERROR"	M 181.1	BOOL	// Fehlermeldung CNC
"APX_PROG_STOP"	M 181.2	BOOL	// Programm Halt
"ApxProgramRun"	M 181.3	BOOL	// Programm läuft
"APX_CNC_READY2RUN"	M 181.4	BOOL	// CNC-Betriebsbereit
"APX_ZPS_BLOW_OUT"	M 181.5	BOOL	// Nullpunktspannsystem Blasluft (Reinigung)
"APX_ZPS_STATUS"	M 181.6	BOOL	// Nullpunktspannsystem Statusmeldung Betriebsartenanzeige (gespannt/gelöst)
"APX_ZPS_RELEASE1"	M 181.7	BOOL	// Nullpunktspannsystem lösen (Ventil_1)
"APX_ZPS_RELEASE2"	M 182.0	BOOL	// Nullpunktspannsystem lösen (Ventil_2)
"APX_SPINDLE_RUN"	M 182.1	BOOL	// Spindel läuft
"APX_CYCLE_START"	M 182.2	BOOL	// Zyklusstart (grüne Starttaste)
"APX_FUNKTION_M20"	M 182.3	BOOL	// Allgemeine Funktion M20
"APX_ZPS_INTERLOCK1"	M 182.4	BOOL	// Nullpunktspannsystem - Ansteuerung (Ventil) für Verriegelungskontrolle
"APX_ZPS_DISTANCE_CHECK1"	M 182.5	BOOL	// Nullpunktspannsystem - Ansteuerung (Ventil) für Auflagenkontrolle
"APX_WORKPIECE_COUNT"	M 182.6	BOOL	// Werkstück Zählimpuls
"APX_PRODUCTION"	M 182.7	BOOL	// Produktionssignal der Werkzeugmaschine/Maschine Produziert (Programm läuft)
"APX_PALLET-NR_BIT0"	M 183.0	BOOL	// Nummer der Palette Arbeitsraum 2^0 (=1)
"APX_PALLET-NR_BIT1"	M 183.1	BOOL	// Nummer der Palette Arbeitsraum 2^1 (=2)
"APX_PALLET-NR_BIT2"	M 183.2	BOOL	// Nummer der Palette Arbeitsraum 2^2 (=4)
"APX_PALLET-NR_BIT3"	M 183.3	BOOL	// Nummer der Palette Arbeitsraum 2^3 (=8)
"APX_ALARM_LIGHT"	M 183.4	BOOL	// Optische Anzeige einer Fehlermeldung
"APX_AUDIBLE_ALARM"	M 183.5	BOOL	// Akustische Ausgabe einer Fehlermeldung
"APX_VCS_RELEASE_FIXTURE1"	M 183.6	BOOL	// Vakuumspannsystem im Arbeitsraum Lösen (=drucklos)
"APX_VCS_RELEASE_FIXTURE2"	M 183.7	BOOL	// Vakuumspannsystem am Rüstplatz Lösen (=drucklos)
"APX_EXH_ON1"	M 184.0	BOOL	// Aktivieren und evtl.verzögertes Abschalten des Nebelabscheiders_1
"APX_COO_COOLANT1_(M8)"	M 184.1	BOOL	// Aktivierung Kühlschmierstoffzufuhr_1 (externe - Spritzdüsen)
"APX_COO_PALLET_CARRIER"	M 184.2	BOOL	// Aktivierung Spänespülung Palettenträger (Umschaltung IKZ)
"APX_COO_WORKPIECE_1"	M 184.3	BOOL	// Aktivierung Spänespülung Werkstückreinigung (Dachspülung - Palettenwechsler)
"APX_COO_SPRAYGUN"	M 184.4	BOOL	// Aktivierung Spritzpistole, Spülpistole
"APX_COO_WORKROOMDOOR"	M 184.5	BOOL	// Aktivierung Spänespülung Kabinentüre, Arbeitsraumtüre
"APX_COO_COOLANT2.2"	M 184.6	BOOL	// Aktivierung Kühlschmierstoffzufuhr_2 (IKZ) - Druckstufe_2
"APX_COO_MAINVALVE"	M 184.7	BOOL	// Aktivierung Kühlschmierstoffzufuhr Haupt-/Zentralventil
"APX_COO_LOCKVALVE_RET"	M 185.0	BOOL	// Aktivierung Sperrventil für Kühlschmierstoffrückführung aus Sammelbehälter (SPF)
"APX_ALARM_RESET"	M 185.1	BOOL	// Bei Betätigung der "Alarm-Quit-Taste (F10)" wird Ausgang gesetzt
"APX_NO_MACHINING"	M 185.2	BOOL	// MDE/BDE: keine Bearbeitung
"APX_INTO_PRODUCTION"	M 185.3	BOOL	// MDE/BDE: Produktionssignal
"ApxProgramEnd"	M 185.4	BOOL	// Programm Ende
"APX_CS_SYST.PRESS1_1"	M 185.5	BOOL	// Spannsystem Systemdruck für Arbeitsraum (Spannkreis 1/Stufe 1)
"APX_CS_RELEASE1_2"	M 185.6	BOOL	// Spannsystem lösen im Arbeitsraum (Spannkreis 1/Stufe 2 - Lösedruck)
"APX_CS_CLAMP1_2"	M 185.7	BOOL	// Spannsystem spannen im Arbeitsraum (Spannkreis 1/Stufe 2 - Spanndruck)
"APX_COO_LOCKVALVE2.2"	M 188.0	BOOL	// Aktivierung Sperrventil für Kühlschmierstoffzufuhr - Druckstufe_2
"APX_CS_BLOW_OUT1_1"	M 188.1	BOOL	// Spannsystem Reinigungsluft im Arbeitsraum (Spannkreis 1 - Blasluft)
"APX_CS_RELEASED1"	M 188.2	BOOL	// Spannsystem im Arbeitsraum gelöst
"APX_CS_CLAMPED1"	M 188.3	BOOL	// Spannsystem im Arbeitsraum gespannt
"APX_CS_STATUS1"	M 188.4	BOOL	// Spannsystem Spannkreis 1 Status/Betriebsmodus (Blink- und Dauersignal)
"APX_EXH_ON2"	M 188.5	BOOL	// Aktivieren und evtl.verzögertes Abschalten des Nebelabscheiders_2
"APX_MCS_STATUS1"	M 188.6	BOOL	// Magnetspannsystem_1 Statusanzeige (Gespannt/gelöst)
"APX_MCS_MODE_ON1"	M 188.7	BOOL	// Magnetspannsystem_1 Anwahl/Aktivierung
"APX_MCS_CLAMPED1"	M 189.0	BOOL	// Magnetspannsystem_1 gespannt
"APX_MCS_RELEASED1"	M 189.1	BOOL	// Magnetspannsystem_1 gelöst
"APX_AXIS_MOVEMENT"	M 189.2	BOOL	// mindestens eine Achse in Bewegung
"APX_APC_ACTIVE"	M 189.3	BOOL	// Palettenwechsel ist aktiv
"APX_TOOL_CHANGE_ACTIVE"	M 189.4	BOOL	// Werkzeugwechsel ist aktiv
"APX_COO_COOLANT2.1"	M 189.5	BOOL	// Aktivierung Kühlschmierstoffzufuhr_2 (IKZ) - Druckstufe_1
"APX_PALLET-NR1_WORKROOM"	M 189.6	BOOL	// Palette_1 im Arbeitsraum
"APX_PALLET-NR2_WORKROOM"	M 189.7	BOOL	// Palette_2 im Arbeitsraum
"APX_PALLET-NR3_WORKROOM"	M 190.0	BOOL	// Palette_3 im Arbeitsraum
"APX_PALLET-NR4_WORKROOM"	M 190.1	BOOL	// Palette_4 im Arbeitsraum
"APX_PALLET-NR5_WORKROOM"	M 190.2	BOOL	// Palette_5 im Arbeitsraum
"APX_PALLET-NR6_WORKROOM"	M 190.3	BOOL	// Palette_6 im Arbeitsraum
"APX_SET-UP"	M 190.4	BOOL	// Rüstvorgang, Rüsten
"APX_FEEDRATE_EQUAL_VALUE"	M 190.5	BOOL	// Position des Vorschubpotentiometers = Wert
"APX_CS_ROTATE_POS0"	M 190.6	BOOL	// Spannvorrichtung - drehen auf Position 0 (z.B. 0 Grad)
"APX_CS_ROTATE_POS1"	M 190.7	BOOL	// Spannvorrichtung - drehen auf Position 1 (z.B. 180 Grad)
"APX_CS_CHECKFINALPOS0"	M 191.0	BOOL	// Spannvorrichtung - Aktivierung für Endlagenüberwachung Position 0
"APX_CS_CHECKFINALPOS1"	M 191.1	BOOL	// Spannvorrichtung - Aktivierung für Endlagenüberwachung Position 1
"APX_COO_LOCKVALVE2.1"	M 191.2	BOOL	// Aktivierung Sperrventil für Kühlschmierstoffzufuhr - Druckstufe_1
"APX_COO_WORKPIECE_2"	M 191.3	BOOL	// Aktivierung Spänespülung Werkstückreinigung (Dachspülung - Arbeitsraum)
"APX_COO_FLUSHPUMP_1"	M 191.4	BOOL	// Aktivierung Förderpumpe Spänespülung(en)
"APX_VCS_ACTIVATED_1"	M 191.5	BOOL	// Vakuumspannsystem - aktiviert
"APX_VCS_STATUS_1"	M 191.6	BOOL	// Vakuumspannsystem - Statusmeldung
"APX_RAPIDVELOCITY=VALUE"	M 191.7	BOOL	// Position des Eilgangpotentiometers = Wert
"APX_MMS_FILLUNIT_START"	M 192.0	BOOL	// MMS: Versorgungseinheit (Tank) befüllen
"APX_MMS_ON"	M 192.1	BOOL	// MMS: Ein/Aktiviert
"APX_ZPS_CHUCKING_POWER1"	M 192.2	BOOL	// Nullpunktspannsystem nachspannen (=Einzugskraft steigern)
"APX_ZPS_STATUS2"	M 192.3	BOOL	// Nullpunktspannsystem Statusmeldung Betriebsartenanzeige (gelöst/gespannt)
"APX_ZPS_CYL_LIFT"	M 192.4	BOOL	// Nullpunktspannsystem - Ansteuerung Ventil Heben (ausfahren)
"APX_ZPS_CYL_LOWER"	M 192.5	BOOL	// Nullpunktspannsystem - Ansteuerung Ventil Senken (einfahren)
"APX_ZPS_CYL_STATUS1"	M 192.6	BOOL	// Nullpunktspannsystem Statusmeldung Abhebezylinder (ausgefahren)
"APX_ZPS_CYL_STATUS2"	M 192.7	BOOL	// Nullpunktspannsystem Statusmeldung Abhebezylinder (eingefahren)
"ApxStatusLightBlue"	M 193.0	BOOL	// Signalleuchte (Ampel) Element: BLAU (BU)
"ApxFeedOverrideInArea"	M 193.1	BOOL	// Vorschub Override im Bereich zwischen xx% und yy%
"ApxFunctionM86"	M 193.2	BOOL	// maschinenspezifische Funktion (M86)
"ApxFunctionM87"	M 193.3	BOOL	// maschinenspezifische Funktion (M87)
"ApxFunctionM88"	M 193.4	BOOL	// maschinenspezifische Funktion (M88)
"ApxFunctionM89"	M 193.5	BOOL	// maschinenspezifische Funktion (M89)
"APX_MCS_UNLOC_PARKSHUTER"	M 193.6	BOOL	// Magnetspannsystem Klappe Parkstation entriegeln
"APX_MCS_PARKSHUTT_UNLOCK"	M 193.7	BOOL	// Magnetspannsystem Meldung Klappe entriegelt
"APX_MCS_MALE_ACTIVE"	M 194.0	BOOL	// Magnetspannsystem Meldung Stecker aktiv
"APX_MCS_MALE_IN_PARKSTAT"	M 194.1	BOOL	// Magnetspannsystem Meldung Stecker in Parkstation
"ApxCooFeedPumpCentrifuge"	M 194.2	BOOL	// Freigabe für Förderpumpe (Einspeisung) Zentrifuge z.B. Niveauüberwachung
"ApxCooScrapeConveyor"	M 194.3	BOOL	// Kratzförderer/Schlammräumer ein
"ApxLubPumpOn"	M 194.4	BOOL	// NC-Rundtisch Schmierstoffpumpe Ein
"ApxAxisStandstill"	M 194.5	BOOL	// Stillstand der Achsen
"ApxMcsSstClamped"	M 194.6	BOOL	// Magnetspannsystem Rüstplatz gespannt
"ApxMcsSstReleased"	M 194.7	BOOL	// Magnetspannsystem Rüstplatz gelöst
"ApxMcsQuitMalfunction"	M 195.0	BOOL	// Magnetspannsystem Störung Quittierung
"ApxCuWarnmessage"	M 195.1	BOOL	// Warnung von Kühlmittelanlage Leistungschalter Sülpistole, Spänesp.,Feinstb....
"ApxCuErrorMessage"	M 195.2	BOOL	// Fehlermeldung von Kühlmittelanlage
"ApxCaErrorMps"	M 195.3	BOOL	// warnung der Leistungsschalter Kühl-/Heizaggregat
"ApxMainValveSusDoor"	M 195.4	BOOL	// Rüstplatztüre(n) Pneumatik-Systemdruck (Sicherheitsventil)
"ApxCloseSusDoor"	M 195.5	BOOL	// Rüstplatztüre(n) schließen
"ApxOpenSusDoor"	M 195.6	BOOL	// Rüstplatztüre(n) öffnen
"ApxCooMainValveHighPress"	M 195.7	BOOL	// Aktivierung Kühlschmierstoffzufuhr Haupt-/Zentralventil Hochdruckkreis
"ApxCooMainValveLowPress"	M 196.0	BOOL	// Aktivierung Kühlschmierstoffzufuhr Haupt-/Zentralventil Niederdruckkreis
"ApxCooLaserToolMeasurem"	M 196.1	BOOL	// Aktivierung Laserspülung Werkzeugvermessung
"ApxChipConvCountClockw_2"	M 196.2	BOOL	// Aktivierung Zusatzspäneförderer Linkslauf
"ApxChipConvClockwise_2"	M 196.3	BOOL	// Aktivierung Zusatzspäneförderer Rechtslauf
"ApxHydFillLevelMinimum"	M 196.4	BOOL	// Füllstand Hydraulik Minimum unterschritten
"ApxCooHighPressureLetOff"	M 196.5	BOOL	// Kühlschmierstoff aus Hochdruckkreis ableiten
"QpxStopAfterToolbreak"	M 196.6	BOOL	// Maschinenstop bei Werkzeugbruch
"QpxBoostCoolant1_M8"	M 196.7	BOOL	// Druckerhöhungspumpe für äußere Kühlmittelzufuhr (M8)
"QpxFlushSetUpStation"	M 197.0	BOOL	// Spänespülung am Rüstplatz (Spannvorrichtung, Werkstück,..)
"m_AkTime"	MD 12	TIME	// ausgeleseneSysZeitVonTime_tck SFC64
"APW_COO_PRESS_VALUE2.2"	MW 186	WORD	// Sollwertvorgabe für Druckvorwahl Kühlmittel_2 (inner Kühlschmierstoffzufuhr)
"CYCL_EXC"	OB 1	OB 1	// Cycle Execution
"I/O_FLT1"	OB 82	OB 82	// I/O Point Fault 1
"CPU_FLT"	OB 84	OB 84	// CPU Fault
"OBNL_FLT"	OB 85	OB 85	// OB Not Loaded Fault
"RACK_FLT"	OB 86	OB 86	// Loss of Rack Fault
"START"	OB 100	OB 100	// Anlauf OB
"PROG_ERR"	OB 121	OB 121	// Programming Error
"MOD_ERR"	OB 122	OB 122	// Module Access Error
"BLKMOV"	SFC 20	SFC 20	// Copy Variables
"TIME_TCK"	SFC 64	SFC 64	// Time tics of period 10 ms
"t0"	T 0	TIMER	// 840D Grundprg.
"t1"	T 1	TIMER	// 840D Grundprg.
"t2"	T 2	TIMER	// 840D Grundprg.
"t3"	T 3	TIMER	// 840D Grundprg.
"t4"	T 4	TIMER	// 840D Grundprg.
"t5"	T 5	TIMER	// 840D Grundprg.
"t6"	T 6	TIMER	// 840D Grundprg.
"t7"	T 7	TIMER	// 840D Grundprg.
"t8"	T 8	TIMER	// 840D Grundprg.
"t9"	T 9	TIMER	// 840D Grundprg.
"t10"	T 10	TIMER
"tHydFilterWarn"	T 11	TIMER	// se Entprellen Signal Warnung Hydraulikfilter
"tDelayStatus1"	T 12	TIMER	// sa Verzögerungszeit Maschinenstatus BDE Signal_1 (machine in run condition)
"tDelayStatus2"	T 13	TIMER	// sa Verzögerungszeit Maschinenstatus BDE Signal_2 (work piece ready)
"tDelayStatus3"	T 14	TIMER	// sa Verzögerungszeit Maschinenstatus BDE Signal_3 (miscellaneous M86)
"tHydOelLevelMinAlarm"	T 15	TIMER	// se Entprellen Signal Alarm Hydraulik Füllstand Minimum
"tHydOelLevelMinWarn"	T 16	TIMER	// se Entprellen Signal Warnung Hydraulik Füllstand Minimum
"tHydOelTempAlarm"	T 17	TIMER	// se Entprellen Signal Alarm Öltemperatur
"tHydFilterAlarm"	T 18	TIMER	// se Entprellen Signal Alarm Hydraulikfilter
"Hilfs_Timer_9"	T 19	TIMER
"Hilfs_Timer_10"	T 20	TIMER
"Hilfs_Timer_11"	T 21	TIMER
"Hilfs_Timer_12"	T 22	TIMER
"Hilfs_Timer_13"	T 23	TIMER
"tDelayFlowMonitoring"	T 24	TIMER	// Bereitschaftsverzögerungszeit für Strömungsüberwachung
"t_toggle"	T 25	TIMER	// Zeit für FB100 Anzeigeintervall
"Hilfs_Timer_15"	T 26	TIMER
"Hilfs_Timer_16"	T 27	TIMER
"Hilfs_Timer_17"	T 28	TIMER
"Hilfs_Timer_18"	T 29	TIMER
"Hilfs_Timer_19"	T 30	TIMER
"Hilfs_Timer_20"	T 31	TIMER
"UDT_MESSAGE"	UDT 2	UDT 2	// UDT zu DB2 (Datenformat für Meldungen)
"UDT101"	UDT 101	UDT 101
"UDT1010"	UDT 1010	UDT 1010	// UDT für UDT 101
"VAT_IN_dbw0"	VAT 1	
"VAT_IN_dbw2"	VAT 2	
"VAT_IN_dbw4"	VAT 3	
"VAT_IN_dbw6"	VAT 4	
"VAT_IN_dbw10_12"	VAT 5	
"VAT_OUT_dbw2"	VAT 6	
"VAT_OUT_dbw0"	VAT 7	
"VAT_PER"	VAT 8	
"VAT_MESSAGE"	VAT 9		// Meldungen, Alarme
"V_Nps0"	VAT 10		// Nullspannsystem
"V_allg"	VAT 11	
"VAT_IN_MP"	VAT 12	
"V_WSpa"	VAT 13		// Werkstückspannsystem
END_SYMBOL_TABLE

TYPE "UDT_MESSAGE"	// UDT 2
AUTHOR : SPAC_slh
NAME : MSG
VERSION : 0.0
  STRUCT
   ALARM_001 : BOOL ;	//Schaltschranktemperatur zu hoch
   ALARM_002 : BOOL ;	//Schaltschranktemperatur - Grenzwert überschritten
   F003 : BOOL ;	//1-
   F004 : BOOL ;	//1-
   F005 : BOOL ;	//1-
   F006 : BOOL ;	//1-
   F007 : BOOL ;	//1-
   F008 : BOOL ;	//1-
   F009 : BOOL ;	//1-
   F010 : BOOL ;	//1-
   F011 : BOOL ;	//1-
   F012 : BOOL ;	//1-
   F013 : BOOL ;	//1-
   F014 : BOOL ;	//1-
   F015 : BOOL ;	//1-
   F016 : BOOL ;	//1-
   ALARM_017 : BOOL ;	//Nullpunktspannsysten Zeitüberschreitung beim Lösen[1]
   ALARM_018 : BOOL ;	//Nullpunktspannsysten Zeitüberschreitung beim Spannen[1]
   ALARM_019 : BOOL ;	//Nullpunktspannsystem Druck am Druckschalter[1]-Maximum nicht vorhanden
   ALARM_020 : BOOL ;	//Nullpunktspannsystem Druck am Druckschalter[1]-Minimum zu hoch
   ALARM_021 : BOOL ;	//Nullpunktspannsystem Signale an Druckschaltern[1] nicht korrekt (Plausibilität)
   ALARM_022 : BOOL ;	//Nullpunktspannsysten Zeitüberschreitung beim Lösen[2]
   ALARM_023 : BOOL ;	//Nullpunktspannsysten Zeitüberschreitung beim Spannen[2]
   ALARM_024 : BOOL ;	//Nullpunktspannsystem Druck am Druckschalter[2]-Maximum nicht vorhanden
   ALARM_025 : BOOL ;	//Nullpunktspannsystem Druck am Druckschalter[2]-Minimum zu hoch
   ALARM_026 : BOOL ;	//Nullpunktspannsystem Signale an Druckschaltern[2] nicht korrekt (Plausibilität)
   ALARM_027 : BOOL ;	//Nullpunktspannsysten Zeitüberschreitung beim Aktivieren der Auflagenkontrolle
   ALARM_028 : BOOL ;	//Nullpunktspannsysten Zeitüberschreitung beim Abschalten der Auflagenkontrolle
   ALARM_029 : BOOL ;	//Nullpunktspannsystem Staudruck für Auflagenkontrolle nicht vorhanden
   ALARM_030 : BOOL ;	//Nullpunktspannsystem Staudruck für Auflagenkontrolle nicht Minimum
   ALARM_031 : BOOL ;	//Nullpunktspannsystem Signale am Auflagenkontrolle nicht korrekt (Plausibilität)
   ALARM_032 : BOOL ;	//Nullpunktspannsysten Zeitüberschreitung beim Aktivieren der Verriegelungskontr.
   ALARM_033 : BOOL ;	//Nullpunktspannsysten Zeitüberschreitung beim Abschalten der Verriegelungskontr.
   ALARM_034 : BOOL ;	//Nullpunktspannsystem Druck an Verriegelungskontrolle nicht vorhanden
   ALARM_035 : BOOL ;	//Nullpunktspannsystem Druck an Verriegelungskontrolle nicht Minimum
   ALARM_036 : BOOL ;	//Nullpunktspannsystem Signale an Verriegelunkontr. nicht korrekt (Plausibilität)
   ALARM_037 : BOOL ;	//Nullpunktspannsystem nicht korrekt gespannt /Freigabe PW nicht möglich
   ALARM_038 : BOOL ;	//Nullpunktspannsystem nicht korrekt gespannt /Verfahren der Achsen nicht möglich
   ALARM_039 : BOOL ;	//Nullpunktspannsystem Lösen nicht möglich
   F040 : BOOL ;	//1-
   F041 : BOOL ;	//1-
   F042 : BOOL ;	//1-
   F043 : BOOL ;	//1-
   F044 : BOOL ;	//1-
   F045 : BOOL ;	//1-
   F046 : BOOL ;	//1-
   F047 : BOOL ;	//1-
   F048 : BOOL ;	//1-
   ALARM_049 : BOOL ;	//Hydraulikfilter Maschine verschmutzt
   ALARM_050 : BOOL ;	//HYD: Hydrauliktemperatur Maschine überschritten
   ALARM_051 : BOOL ;	//CS: Spannhydraulikfilter Maschine verschmutzt
   F052 : BOOL ;	//1-
   F053 : BOOL ;	//1-
   F054 : BOOL ;	//1-
   F055 : BOOL ;	//1-
   F056 : BOOL ;	//1-
   ALARM_057 : BOOL ;	//MMS: Befülleinheit MMS - kein Öl vorhanden
   ALARM_058 : BOOL ;	//MMS: Ölnebelzerstäuber MMS - kein Öl vorhanden
   ALARM_059 : BOOL ;	//MMS: Ölnebelzerstäuber MMS - Vorwarnung Minimum
   F060 : BOOL ;	//1-
   F061 : BOOL ;	//1-
   F062 : BOOL ;	//1-
   F063 : BOOL ;	//1-
   F064 : BOOL ;	//1-
   ALARM_065 : BOOL ;	//Störung in Energieversorgung Nebel-u.Rauchabscheider_1
   ALARM_066 : BOOL ;	//Störung in Energieversorgung Nebel-u.Rauchabscheider_2
   F067 : BOOL ;	//1-
   F068 : BOOL ;	//1-
   F069 : BOOL ;	//1-
   F070 : BOOL ;	//1-
   F071 : BOOL ;	//1-
   F072 : BOOL ;	//1-
   F073 : BOOL ;	//1-
   F074 : BOOL ;	//1-
   F075 : BOOL ;	//1-
   F076 : BOOL ;	//1-
   F077 : BOOL ;	//1-
   F078 : BOOL ;	//1-
   F079 : BOOL ;	//1-
   F080 : BOOL ;	//1-
   ALARM_081 : BOOL ;	//Vakuumspannsystem Zeitüberschreitung beim Lösen (Arbeitsraum)
   ALARM_082 : BOOL ;	//Vakuumspannsystem Zeitüberschreitung beim Spannen (Arbeitsraum)
   ALARM_083 : BOOL ;	//Vakuumspannsystem Druck am Druckschalter-Maximum nicht vorhanden (Arbeitsraum)
   ALARM_084 : BOOL ;	//Vakuumspannsystem Druck am Druckschalter-Minimum zu hoch (Arbeitsraum)
   ALARM_085 : BOOL ;	//Vakuumspannsystem Signale an Druckschaltern nicht korrekt-Plausibilität (ARB)
   ALARM_086 : BOOL ;	//Vakuumspannsystem im Arbeitsraum nicht Betriebsbereit (z.B.Störung der Energie)
   ALARM_087 : BOOL ;	//Vakuumspannsystem am Rüstplatz nicht Betriebsbereit (z.B.Störung der Energie)
   ALARM_088 : BOOL ;	//Vakuumspannsystem Zeitüberschreitung beim Lösen (Rüstplatz)
   ALARM_089 : BOOL ;	//Vakuumspannsystem Zeitüberschreitung beim Spannen (Rüstplatz)
   ALARM_090 : BOOL ;	//Vakuumspannsystem Druck am Druckschalter-Minimum zu hoch (Rüstplatz)
   ALARM_091 : BOOL ;	//Vakuumspannsystem Druck am Druckschalter-Maximum nicht vorhanden (Rüstplatz)
   ALARM_092 : BOOL ;	//Vakuumspannsystem Signale an Druckschaltern nicht korrekt-Plausibilität (RPL)
   ALARM_093 : BOOL ;	//KSS: Hauptventil in Zuleitung nicht geöffnet (Hochdruckkreis)
   ALARM_094 : BOOL ;	//KSS: Hauptventil in Zuleitung nicht geschlossen (Hochdruckkreis)
   ALARM_095 : BOOL ;	//KSS: Hauptventil in Zuleitung nicht geöffnet (Niederdruckkreis)
   ALARM_096 : BOOL ;	//KSS: Hauptventil in Zuleitung nicht geschlossen (Niderdruckkreis)
   ALARM_097 : BOOL ;	//Km-Hautpventil nicht offen, E9.0 meldet "zu", muss 0-Signal melden
   ALARM_098 : BOOL ;	//Km-Hautpventil schließt nicht, E9.0 muss 1-Signal melden
   ALARM_099 : BOOL ;	//WHG-Alarm
   ALARM_100 : BOOL ;	//minimaler Füllstand in KSA erreicht
   ALARM_101 : BOOL ;	//Km-Systemdruck fehlt, E8.3 muss 1-Signal melden
   ALARM_102 : BOOL ;	//Km-Systemdruck, Druckschalter defekt, E8.3 muss 0-Signal melden
   ALARM_103 : BOOL ;	//Km-Durchfluss fehlt, E9.2 muss 1-Signal melden
   ALARM_104 : BOOL ;	//Km-Durchfluss-Schalter defekt, E9.2 muss 0-Signal melden
   ALARM_105 : BOOL ;	//Kühlmittelfeinfilter verschmutzt E10.1
   ALARM_106 : BOOL ;	//Kühlmittelfeinfilter Schalterpaarüberwachung E10.1/E102
   ALARM_107 : BOOL ;	//KSS: KSS-Druck für Spüleinrichtung nicht erreicht/vorhanden
   ALARM_108 : BOOL ;	//KSS: max. KSS-Druck für Spüleinrichtung überschritten
   ALARM_109 : BOOL ;	//KSS: KSS-Druck für Spüleinrichtung nicht Minimum
   ALARM_110 : BOOL ;	//KSS: Pneumatikdruck an Kühlschmierstoffanlage unterschritten
   ALARM_111 : BOOL ;	//KSS: Maschine-Ein (kein Not-Aus) Signal an Kühlschmierstoffanlage nicht vorh.
   F112 : BOOL ;	//1-
   ALARM_113 : BOOL ;	//Zeitüberschreitung beim Aktivieren der KSS-Zufuhr (Niederdruck)
   ALARM_114 : BOOL ;	//Funktionsüberwachung Strömungssensor - Unterbrechung (Niederdruck)
   ALARM_115 : BOOL ;	//Zeitüberschreitung beim Abschalten der KSS-Zufuhr (Niederdruck)
   ALARM_116 : BOOL ;	//Leitungsüberwachung Strömungssensor (Niederdruck)
   ALARM_117 : BOOL ;	//Zeitüberschreitung beim Aktivieren der KSS-Zufuhr (Hochdruck)
   ALARM_118 : BOOL ;	//Funktionsüberwachung Strömungssensor - Unterbrechung (Hochdruck)
   ALARM_119 : BOOL ;	//Zeitüberschreitung beim Abschalten der KSS-Zufuhr (Hochdruck)
   ALARM_120 : BOOL ;	//Leitungsüberwachung Strömungssensor (Hochdruck)
   ALARM_121 : BOOL ;	//KSS: Systemdruck in Zuleitung fehlt (Hochdruckkreis)
   ALARM_122 : BOOL ;	//KSS: Systemdruck bei abgeschalteter KSS-Zuffuhr vorhanden (Hochdruckkreis)
   ALARM_123 : BOOL ;	//KSS: Systemdruck in Zuleitung fehlt (Niederdruck)
   ALARM_124 : BOOL ;	//KSS: Systemdruck bei abgeschalteter KSS-Zuffuhr vorhanden (Niederdruckkreis)
   ALARM_125 : BOOL ;	//KSS: keine KSS-Strömung bei aktivierter KSS-Zufuhr (Hochdruckkreis)
   ALARM_126 : BOOL ;	//KSS: KSS-Strömung beiabgeschalteter KSS-Zufuhr vorhanden (Hochdruckkreis)
   ALARM_127 : BOOL ;	//KSS: keine KSS-Strömung bei aktivierter KSS-Zufuhr (Niederdruckkreis)
   ALARM_128 : BOOL ;	//KSS: KSS-Strömung beiabgeschalteter KSS-Zufuhr vorhanden (Niederdruckkreis)
   ALARM_129 : BOOL ;	//Spannsystem Zeitüberschreitung beim SysDruck für Lösen aktivieren[1]
   ALARM_130 : BOOL ;	//Spannsystem Zeitüberschreitung beim Spannen[1]
   ALARM_131 : BOOL ;	//Spannsystem Systemdruck für Lösen [1]-Maximum nicht vorhanden
   ALARM_132 : BOOL ;	//Spannsystem Systemdruck für Lösen [1]-Minimum,Restdruck vorhanden
   ALARM_133 : BOOL ;	//Spannsystem Signale an Druckschaltern[1] nicht korrekt (Plausibilität)
   ALARM_134 : BOOL ;	//Spannsystem Zeitüberschreitung beim Lösen[2]
   ALARM_135 : BOOL ;	//Spannsystem Zeitüberschreitung beim Spannen[2]
   ALARM_136 : BOOL ;	//Spannsystem nicht gelöst[2], Endlage verlassen
   ALARM_137 : BOOL ;	//Spannsystem nicht gespannt[2], Endlage verlassen
   ALARM_138 : BOOL ;	//Spannsystem Signale an Druckschaltern[2] nicht korrekt (Plausibilität)
   ALARM_139 : BOOL ;	//Spannsystem Zeitüberschreitung beim Aktivieren der Auflagenkontrolle
   ALARM_140 : BOOL ;	//Spannsystem Zeitüberschreitung beim Abschalten der Auflagenkontrolle
   ALARM_141 : BOOL ;	//Spannsystem Staudruck für Auflagenkontrolle nicht vorhanden
   ALARM_142 : BOOL ;	//Spannsystem Staudruck für Auflagenkontrolle nicht Minimum
   ALARM_143 : BOOL ;	//Spannsystem Signale am Auflagenkontrolle nicht korrekt (Plausibilität)
   ALARM_144 : BOOL ;	//Spannsystem spannen mit Wkst.aber Schalter "gespannt ohne Wkst"=log.1
   ALARM_145 : BOOL ;	//Spannsystem Schalterpaarüberwachung gelöst:Druck vorhanden/drucklos
   ALARM_146 : BOOL ;	//Spannsystem Schalterpaarüberwachung gespannt:Druck vorhanden/drucklos
   ALARM_147 : BOOL ;	//Spannsystem Endlage der Spannvorrichtung nicht erreicht (Drehbewegung Pos.0)
   ALARM_148 : BOOL ;	//Spannsystem Endlage der Spannvorrichtung nicht erreicht (Drehbewegung Pos.1)
   ALARM_149 : BOOL ;	//Spannvorrichtung hydr. Systemdruck für Drehbwewegung Pos 0 nicht vorhanden
   ALARM_150 : BOOL ;	//Spannvorrichtung hydr. Systemdruck für Drehbwewegung Pos 1 nicht vorhanden
   ALARM_151 : BOOL ;	//Schlüsselschalter für Spannhydraulik "AUS"
   ALARM_152 : BOOL ;	//Spannvorrichtung: Schalterpaarüberwachung Hydraulik
   ALARM_153 : BOOL ;	//Spannvorrichtung: Schalterpaarüberwachung Pneumatik
   F154 : BOOL ;	//1-
   F155 : BOOL ;	//1-
   F156 : BOOL ;	//1-
   F157 : BOOL ;	//1-
   F158 : BOOL ;	//1-
   F159 : BOOL ;	//1-
   F160 : BOOL ;	//1-
   ALARM_161 : BOOL ;	//Magnetspannsystem nicht korrekt gespannt /Freigabe PW nicht möglich
   ALARM_162 : BOOL ;	//Magnetspannsystem Steckverbindung nicht in Ablagevorrichtung
   ALARM_163 : BOOL ;	//Magnetspannsystem Werkstück am Rüstplatz nicht korrekt gespannt
   ALARM_164 : BOOL ;	//Magnetspannsystem Werkstück im Arbeitsraum nicht korrekt gespannt
   F165 : BOOL ;	//1-
   F166 : BOOL ;	//1-
   F167 : BOOL ;	//1-
   F168 : BOOL ;	//1-
   F169 : BOOL ;	//1-
   F170 : BOOL ;	//1-
   F171 : BOOL ;	//1-
   F172 : BOOL ;	//1-
   F173 : BOOL ;	//1-
   F174 : BOOL ;	//1-
   F175 : BOOL ;	//1-
   F176 : BOOL ;	//1-
   ALARM_177 : BOOL ;	//Kameraüberwachung angesprochen
   ALARM_178 : BOOL ;	//Störung Löschanlage
   ALARM_179 : BOOL ;	//Störung Kühlmittelanlage
   F180 : BOOL ;	//1-
   F181 : BOOL ;	//1-
   F182 : BOOL ;	//1-
   F183 : BOOL ;	//1-
   F184 : BOOL ;	//1-
   F185 : BOOL ;	//1-
   F186 : BOOL ;	//1-
   F187 : BOOL ;	//1-
   F188 : BOOL ;	//1-
   F189 : BOOL ;	//1-
   F190 : BOOL ;	//1-
   F191 : BOOL ;	//1-
   F192 : BOOL ;	//1-
   ALARM_193 : BOOL ;	//LUB: Druck an Schmierverteiler Querachse nicht erreicht
   ALARM_194 : BOOL ;	//LUB: Zeitüberschreitung beim Abschalten der Schmierung (Querachse)
   ALARM_195 : BOOL ;	//LUB: Druck an Schmierverteiler Längsachse nicht erreicht
   ALARM_196 : BOOL ;	//LUB: Zeitüberschreitung beim Abschalten der Schmierung (Längsachse)
   ALARM_197 : BOOL ;	//LUB: Druck an Schmierverteiler Vertikalachse nicht erreicht
   ALARM_198 : BOOL ;	//LUB: Zeitüberschreitung beim Abschalten der Schmierung (Vertikalachse)
   ALARM_199 : BOOL ;	//LUB: Druck an Schmierverteiler des Palettenwechsler nicht erreicht
   ALARM_200 : BOOL ;	//LUB: Zeitüberschreitung beim Abschalten der Schmierung (Palettenwechsler)
   ALARM_201 : BOOL ;	//LUB: Druck an Schmierverteiler des Werkzeugmagazin-/wechsler nicht erreicht
   ALARM_202 : BOOL ;	//LUB: Zeitüberschreitung beim Abschalten der Schmierung (Werkzeugmagazin-/wech)
   ALARM_203 : BOOL ;	//LUB: Druck an Schmierverteiler des Rüstplatzes nicht erreicht
   ALARM_204 : BOOL ;	//LUB: Zeitüberschreitung beim Abschalten der Schmierung (Rüstplatzes)
   ALARM_205 : BOOL ;	//LUB: Druck an Schmierverteiler Querachse_1 nicht erreicht
   ALARM_206 : BOOL ;	//LUB: Zeitüberschreitung beim Abschalten der Schmierung (Querachse_1)
   ALARM_207 : BOOL ;	//LUB: Druck an Schmierverteiler Längsachse_1 nicht erreicht
   ALARM_208 : BOOL ;	//LUB: Zeitüberschreitung beim Abschalten der Schmierung (Längsachse_1)
   ALARM_209 : BOOL ;	//LUB: Druck an Schmierverteiler NC-Rundtisch nicht erreicht
   ALARM_210 : BOOL ;	//LUB: Zeitüberschreitung beim Abschalten der Schmierung (NC-Rundtisch)
   F211 : BOOL ;	//1-
   F212 : BOOL ;	//1-
   F213 : BOOL ;	//1-
   F214 : BOOL ;	//1-
   F215 : BOOL ;	//1-
   F216 : BOOL ;	//1-
   ALARM_217 : BOOL ;	//Systemdruck (Pneumatik) Antrieb Rüstplatztüre(n) nicht vorhanden
   ALARM_218 : BOOL ;	//Zeitüberschreitung beim Abschalten des Systemdruckes autom.Rüstplatztüre(n)
   ALARM_219 : BOOL ;	//Die Endlage "offen" der linken Rüstplatztüre wurde verlassen
   ALARM_220 : BOOL ;	//Die Endlage "geschlossen" der linken Rüstplatztüre wurde verlassen
   ALARM_221 : BOOL ;	//Plausibilitätsüberwachung der Endschalter "Rüstplatztüre links"
   ALARM_222 : BOOL ;	//Die Endlage "offen" der rechten Rüstplatztüre wurde verlassen
   ALARM_223 : BOOL ;	//Die Endlage "geschlossen" der rechten Rüstplatztüre wurde verlassen
   ALARM_224 : BOOL ;	//Plausibilitätsüberwachung der Endschalter "Rüstplatztüre rechts"
   ALARM_225 : BOOL ;	//Drucküberwachung Rüstplatztüre(n) öffnen - benötigter Druck nicht vorhanden
   ALARM_226 : BOOL ;	//Drucküberwachung Rüstplatztüre(n) öffnen - Zeitüberschreitung beim Abschalten
   ALARM_227 : BOOL ;	//Drucküberwachung Rüstplatztüre(n) schliessen - benötigter Druck nicht vorhanden
   ALARM_228 : BOOL ;	//Drucküberwachung Rüstplatztüre(n) schliessen - Zeitüberschreitung b. Abschalten
   F229 : BOOL ;	//1-
   F230 : BOOL ;	//1-
   F231 : BOOL ;	//1-
   F232 : BOOL ;	//1-
   ALARM_233 : BOOL ;	//Schaltleiste an Rüstplatztüre(n) wurde betätigt - automatischer Rücklauf
   ALARM_234 : BOOL ;	//Schaltleiste an Rüstplatztüre(n) wurde betätigt
   F235 : BOOL ;	//1-
   F236 : BOOL ;	//1-
   F237 : BOOL ;	//1-
   F238 : BOOL ;	//1-
   F239 : BOOL ;	//1-
   F240 : BOOL ;	//1-
   F241 : BOOL ;	//1-
   F242 : BOOL ;	//1-
   F243 : BOOL ;	//1-
   F244 : BOOL ;	//1-
   F245 : BOOL ;	//1-
   F246 : BOOL ;	//1-
   F247 : BOOL ;	//1-
   F248 : BOOL ;	//1-
   F249 : BOOL ;	//1-
   F250 : BOOL ;	//1-
   F251 : BOOL ;	//1-
   F252 : BOOL ;	//1-
   F253 : BOOL ;	//1-
   F254 : BOOL ;	//1-
   F255 : BOOL ;	//1-
   F256 : BOOL ;	//1-
   F257 : BOOL ;	//1-
   F258 : BOOL ;	//1-
   F259 : BOOL ;	//1-
   F260 : BOOL ;	//1-
   F261 : BOOL ;	//1-
   F262 : BOOL ;	//1-
   F263 : BOOL ;	//1-
   F264 : BOOL ;	//1-
   F265 : BOOL ;	//1-
   F266 : BOOL ;	//1-
   F267 : BOOL ;	//1-
   F268 : BOOL ;	//1-
   F269 : BOOL ;	//1-
   F270 : BOOL ;	//1-
   F271 : BOOL ;	//1-
   F272 : BOOL ;	//1-
   F273 : BOOL ;	//1-
   F274 : BOOL ;	//1-
   F275 : BOOL ;	//1-
   F276 : BOOL ;	//1-
   F277 : BOOL ;	//1-
   F278 : BOOL ;	//1-
   F279 : BOOL ;	//1-
   F280 : BOOL ;	//1-
   F281 : BOOL ;	//1-
   F282 : BOOL ;	//1-
   F283 : BOOL ;	//1-
   F284 : BOOL ;	//1-
   F285 : BOOL ;	//1-
   F286 : BOOL ;	//1-
   F287 : BOOL ;	//1-
   F288 : BOOL ;	//1-
   F289 : BOOL ;	//1-
   F290 : BOOL ;	//1-
   F291 : BOOL ;	//1-
   F292 : BOOL ;	//1-
   F293 : BOOL ;	//1-
   F294 : BOOL ;	//1-
   F295 : BOOL ;	//1-
   F296 : BOOL ;	//1-
   F297 : BOOL ;	//1-
   F298 : BOOL ;	//1-
   F299 : BOOL ;	//1-
   F300 : BOOL ;	//1-
   F301 : BOOL ;	//1-
   F302 : BOOL ;	//1-
   F303 : BOOL ;	//1-
   F304 : BOOL ;	//1-
   F305 : BOOL ;	//1-
   F306 : BOOL ;	//1-
   F307 : BOOL ;	//1-
   F308 : BOOL ;	//1-
   F309 : BOOL ;	//1-
   F310 : BOOL ;	//1-
   F311 : BOOL ;	//1-
   F312 : BOOL ;	//1-
   F313 : BOOL ;	//1-
   F314 : BOOL ;	//1-
   F315 : BOOL ;	//1-
   F316 : BOOL ;	//1-
   F317 : BOOL ;	//1-
   F318 : BOOL ;	//1-
   F319 : BOOL ;	//1-
   F320 : BOOL ;	//1-
   F321 : BOOL ;	//1-
   F322 : BOOL ;	//1-
   F323 : BOOL ;	//1-
   F324 : BOOL ;	//1-
   F325 : BOOL ;	//1-
   F326 : BOOL ;	//1-
   F327 : BOOL ;	//1-
   F328 : BOOL ;	//1-
   F329 : BOOL ;	//1-
   F330 : BOOL ;	//1-
   F331 : BOOL ;	//1-
   F332 : BOOL ;	//1-
   F333 : BOOL ;	//1-
   F334 : BOOL ;	//1-
   F335 : BOOL ;	//1-
   F336 : BOOL ;	//1-
   F337 : BOOL ;	//1-
   F338 : BOOL ;	//1-
   F339 : BOOL ;	//1-
   F340 : BOOL ;	//1-
   F341 : BOOL ;	//1-
   F342 : BOOL ;	//1-
   F343 : BOOL ;	//1-
   F344 : BOOL ;	//1-
   F345 : BOOL ;	//1-
   F346 : BOOL ;	//1-
   F347 : BOOL ;	//1-
   F348 : BOOL ;	//1-
   F349 : BOOL ;	//1-
   F350 : BOOL ;	//1-
   F351 : BOOL ;	//1-
   F352 : BOOL ;	//1-
   F353 : BOOL ;	//1-
   F354 : BOOL ;	//1-
   F355 : BOOL ;	//1-
   F356 : BOOL ;	//1-
   F357 : BOOL ;	//1-
   F358 : BOOL ;	//1-
   F359 : BOOL ;	//1-
   F360 : BOOL ;	//1-
   F361 : BOOL ;	//1-
   F362 : BOOL ;	//1-
   F363 : BOOL ;	//1-
   F364 : BOOL ;	//1-
   F365 : BOOL ;	//1-
   F366 : BOOL ;	//1-
   F367 : BOOL ;	//1-
   F368 : BOOL ;	//1-
   F369 : BOOL ;	//1-
   F370 : BOOL ;	//1-
   F371 : BOOL ;	//1-
   F372 : BOOL ;	//1-
   F373 : BOOL ;	//1-
   F374 : BOOL ;	//1-
   F375 : BOOL ;	//1-
   F376 : BOOL ;	//1-
   F377 : BOOL ;	//1-
   F378 : BOOL ;	//1-
   F379 : BOOL ;	//1-
   F380 : BOOL ;	//1-
   F381 : BOOL ;	//1-
   F382 : BOOL ;	//1-
   F383 : BOOL ;	//1-
   F384 : BOOL ;	//1-
   F385 : BOOL ;	//1-
   F386 : BOOL ;	//1-
   F387 : BOOL ;	//1-
   F388 : BOOL ;	//1-
   F389 : BOOL ;	//1-
   F390 : BOOL ;	//1-
   F391 : BOOL ;	//1-
   F392 : BOOL ;	//1-
   F393 : BOOL ;	//1-
   F394 : BOOL ;	//1-
   F395 : BOOL ;	//1-
   F396 : BOOL ;	//1-
   F397 : BOOL ;	//1-
   F398 : BOOL ;	//1-
   F399 : BOOL ;	//1-
   F400 : BOOL ;	//1-
   F401 : BOOL ;	//1-
   F402 : BOOL ;	//1-
   F403 : BOOL ;	//1-
   F404 : BOOL ;	//1-
   F405 : BOOL ;	//1-
   F406 : BOOL ;	//1-
   F407 : BOOL ;	//1-
   F408 : BOOL ;	//1-
   F409 : BOOL ;	//1-
   F410 : BOOL ;	//1-
   F411 : BOOL ;	//1-
   F412 : BOOL ;	//1-
   F413 : BOOL ;	//1-
   F414 : BOOL ;	//1-
   F415 : BOOL ;	//1-
   F416 : BOOL ;	//1-
   F417 : BOOL ;	//1-
   F418 : BOOL ;	//1-
   F419 : BOOL ;	//1-
   F420 : BOOL ;	//1-
   F421 : BOOL ;	//1-
   F422 : BOOL ;	//1-
   F423 : BOOL ;	//1-
   F424 : BOOL ;	//1-
   F425 : BOOL ;	//1-
   F426 : BOOL ;	//1-
   F427 : BOOL ;	//1-
   F428 : BOOL ;	//1-
   F429 : BOOL ;	//1-
   F430 : BOOL ;	//1-
   F431 : BOOL ;	//1-
   F432 : BOOL ;	//1-
   F433 : BOOL ;	//1-
   F434 : BOOL ;	//1-
   F435 : BOOL ;	//1-
   F436 : BOOL ;	//1-
   F437 : BOOL ;	//1-
   F438 : BOOL ;	//1-
   F439 : BOOL ;	//1-
   F440 : BOOL ;	//1-
   F441 : BOOL ;	//1-
   F442 : BOOL ;	//1-
   F443 : BOOL ;	//1-
   F444 : BOOL ;	//1-
   F445 : BOOL ;	//1-
   F446 : BOOL ;	//1-
   F447 : BOOL ;	//1-
   F448 : BOOL ;	//1-
   F449 : BOOL ;	//1-
   F450 : BOOL ;	//1-
   F451 : BOOL ;	//1-
   F452 : BOOL ;	//1-
   F453 : BOOL ;	//1-
   F454 : BOOL ;	//1-
   F455 : BOOL ;	//1-
   F456 : BOOL ;	//1-
   F457 : BOOL ;	//1-
   F458 : BOOL ;	//1-
   F459 : BOOL ;	//1-
   F460 : BOOL ;	//1-
   F461 : BOOL ;	//1-
   F462 : BOOL ;	//1-
   F463 : BOOL ;	//1-
   F464 : BOOL ;	//1-
   F465 : BOOL ;	//1-
   F466 : BOOL ;	//1-
   F467 : BOOL ;	//1-
   F468 : BOOL ;	//1-
   F469 : BOOL ;	//1-
   F470 : BOOL ;	//1-
   F471 : BOOL ;	//1-
   F472 : BOOL ;	//1-
   F473 : BOOL ;	//1-
   F474 : BOOL ;	//1-
   F475 : BOOL ;	//1-
   F476 : BOOL ;	//1-
   F477 : BOOL ;	//1-
   F478 : BOOL ;	//1-
   F479 : BOOL ;	//1-
   F480 : BOOL ;	//1-
   F481 : BOOL ;	//1-
   F482 : BOOL ;	//1-
   F483 : BOOL ;	//1-
   F484 : BOOL ;	//1-
   F485 : BOOL ;	//1-
   F486 : BOOL ;	//1-
   F487 : BOOL ;	//1-
   F488 : BOOL ;	//1-
   F489 : BOOL ;	//1-
   F490 : BOOL ;	//1-
   F491 : BOOL ;	//1-
   F492 : BOOL ;	//1-
   F493 : BOOL ;	//1-
   F494 : BOOL ;	//1-
   F495 : BOOL ;	//1-
   F496 : BOOL ;	//1-
   F497 : BOOL ;	//1-
   F498 : BOOL ;	//1-
   F499 : BOOL ;	//1-
   F500 : BOOL ;	//1-
   F501 : BOOL ;	//1-
   F502 : BOOL ;	//1-
   F503 : BOOL ;	//1-
   F504 : BOOL ;	//1-
   F505 : BOOL ;	//1-
   F506 : BOOL ;	//1-
   F507 : BOOL ;	//1-
   F508 : BOOL ;	//1-
   F509 : BOOL ;	//1-
   ALARM_510 : BOOL ;	//Meldung Kameraüberwachung
   ALARM_511 : BOOL ;	//Meldung Löschanlage
   F512 : BOOL ;	//1-
   MSG_513 : BOOL ;	//Schaltschranktüre(n) an Werkzeugmaschine geöffnet
   MSG_514 : BOOL ;	//Schaltschranktüre(n) an Kühlschmierstoffanlage geöffnet
   MSG_515 : BOOL ;	//Schaltschranktemperatur zu hoch
   Me516 : BOOL ;	//1-
   Me517 : BOOL ;	//1-
   Me518 : BOOL ;	//1-
   Me519 : BOOL ;	//1-
   Me520 : BOOL ;	//1-
   Me521 : BOOL ;	//1-
   Me522 : BOOL ;	//1-
   Me523 : BOOL ;	//1-
   Me524 : BOOL ;	//1-
   Me525 : BOOL ;	//1-
   Me526 : BOOL ;	//1-
   Me527 : BOOL ;	//1-
   MSG_528 : BOOL ;	//CS: Spannhydraulikfilter Maschine verschmutzt
   MSG_529 : BOOL ;	//Hydraulikfilter Maschine verschmutzt
   MSG_530 : BOOL ;	//HYD:Hydraulik Maschine Füllstand Maximum überschritten
   MSG_531 : BOOL ;	//HYD:Hydraulik Maschine Füllstand Minimum unterschritten
   Me532 : BOOL ;	//1-
   Me533 : BOOL ;	//1-
   Me534 : BOOL ;	//1-
   Me535 : BOOL ;	//1-
   Me536 : BOOL ;	//1-
   Me537 : BOOL ;	//1-
   Me538 : BOOL ;	//1-
   Me539 : BOOL ;	//1-
   Me540 : BOOL ;	//1-
   Me541 : BOOL ;	//1-
   Me542 : BOOL ;	//1-
   Me543 : BOOL ;	//1-
   Me544 : BOOL ;	//1-
   MSG_545 : BOOL ;	//Vakuumspannsystem nicht gespannt (Arbeitsraum)
   MSG_546 : BOOL ;	//Vakuumspannsystem nicht gespannt (Rüstplatz)
   MSG_547 : BOOL ;	//Vakuumspannsystem: Lösen nicht möglich
   Me548 : BOOL ;	//1-
   Me549 : BOOL ;	//1-
   Me550 : BOOL ;	//1-
   Me551 : BOOL ;	//1-
   Me552 : BOOL ;	//1-
   Me553 : BOOL ;	//1-
   Me554 : BOOL ;	//1-
   Me555 : BOOL ;	//1-
   Me556 : BOOL ;	//1-
   Me557 : BOOL ;	//1-
   Me558 : BOOL ;	//1-
   Me559 : BOOL ;	//1-
   Me560 : BOOL ;	//1-
   MSG_561 : BOOL ;	//KSS: Warnung von Kühlschmierstoffanlage
   MSG_562 : BOOL ;	//KSS: Warnung! Feinfilter Kühlschmierstoffanlage verschmutzt
   MSG_563 : BOOL ;	//KSS: Die gewählte Druckstufe liegt nicht im möglichen Wertebereich!
   MSG_564 : BOOL ;	//KSS: Störung der Energieversorgung Zentrifuge
   MSG_565 : BOOL ;	//KSS: Vorwarnung Füllstand Kühlschmierstoff im Feinbereich
   MSG_566 : BOOL ;	//KSS: Funktionsstörung der Zentrifuge
   MSG_567 : BOOL ;	//KSS: Reinigungsintervall für Zentrifuge
   MSG_568 : BOOL ;	//KSS: Grenzwert in Kühlschmierstoffanlage überschritten (WHG)
   MSG_569 : BOOL ;	//KSS: Grobpartikel Doppelfilter verschmutzt
   Me570 : BOOL ;	//1-
   Me571 : BOOL ;	//1-
   Me572 : BOOL ;	//1-
   Me573 : BOOL ;	//1-
   Me574 : BOOL ;	//1-
   Me575 : BOOL ;	//1-
   MSG_576 : BOOL ;	//Störung an externer Späneentsorgung
   MSG_577 : BOOL ;	//Löseanforderung von extern aber keine Freigabe von LeitPLC
   MSG_578 : BOOL ;	//Löseanforderung aber Spannsystem nicht aktiviert
   MSG_579 : BOOL ;	//Nullpunktspannsstem ist gelöst
   Me580 : BOOL ;	//1-
   Me581 : BOOL ;	//1-
   Me582 : BOOL ;	//1-
   Me583 : BOOL ;	//1-
   Me584 : BOOL ;	//1-
   Me585 : BOOL ;	//1-
   Me586 : BOOL ;	//1-
   Me587 : BOOL ;	//1-
   Me588 : BOOL ;	//1-
   Me589 : BOOL ;	//1-
   Me590 : BOOL ;	//1-
   Me591 : BOOL ;	//1-
   Me592 : BOOL ;	//1-
   MSG_593 : BOOL ;	//Vorwarnung min. Füllstand Behälter MMS
   MSG_594 : BOOL ;	//min.Füllstand in Versorgungseinheit MMS unterschritten
   Me595 : BOOL ;	//1-
   Me596 : BOOL ;	//1-
   Me597 : BOOL ;	//1-
   Me598 : BOOL ;	//1-
   Me599 : BOOL ;	//1-
   MSG_600 : BOOL ;	//NOT-AUS Bedienpult betätigt
   MSG_601 : BOOL ;	//NOT-AUS Bedienpult Handrad betätigt
   MSG_602 : BOOL ;	//NOT-AUS Späneförderer betätigt
   MSG_603 : BOOL ;	//NOT-AUS Werkzeugeingabestation betätigt
   MSG_604 : BOOL ;	//NOT-AUS Rüstplatz betätigt
   MSG_605 : BOOL ;	//NOT-AUS Werkzeugmagazin Handrad betätigt
   MSG_606 : BOOL ;	//NOT-Aus Werkzeugmagazin
   Me607 : BOOL ;	//1-
   Me608 : BOOL ;	//1-
   Me609 : BOOL ;	//1-
   Me610 : BOOL ;	//1-
   MSG_611 : BOOL ;	//Leitungsschutzschalter Steckdose Frontschild hat ausgelöst
   MSG_612 : BOOL ;	//Leitungsschutzschalter Schmierstoffpumpe hat ausgelöst
   MSG_613 : BOOL ;	//Leitungsschutzschalter AS-i Netzteil hat ausgelöst
   MSG_614 : BOOL ;	//Leitungsschutzschalter Durchflussüberwachung hat ausgelöst
   MSG_615 : BOOL ;	//Leitungsschutzschalter Leuchtmelder Kommandostation hat ausgelöst
   MSG_616 : BOOL ;	//Leitungsschutzschalter Steuerstromkreis hat ausgelöst
   MSG_617 : BOOL ;	//Leitungsschutzschalter CNC-Steuerung hat ausgelöst
   MSG_618 : BOOL ;	//Leitungsschutzschalter Not-Aus Steuerstromkreis hat ausgelöst
   MSG_619 : BOOL ;	//Leitungsschutzschalter Werkzeugwechsler hat ausgelöst
   MSG_620 : BOOL ;	//Leitungsschutzschalter DC-Steuerspannung hat ausgelöst
   MSG_621 : BOOL ;	//Leitungsschutzschalter Palettenwechsler hat ausgelöst
   MSG_622 : BOOL ;	//Leitungsschutzschalter Kühlmittelanlage hat ausgelöst
   MSG_623 : BOOL ;	//Leitungsschutzschalter PCU 50 hat ausgelöst
   MSG_624 : BOOL ;	//Leitungsschutzschalter Bildschirm hat ausgelöst
   MSG_625 : BOOL ;	//Leitungsschutzschalter IM151 Maschine hat ausgelöst
   MSG_626 : BOOL ;	//Leitungsschutzschalter_1 Ausgänge IM151 hat ausgelöst
   MSG_627 : BOOL ;	//Leitungsschutzschalter_2 Ausgänge IM151 hat ausgelöst
   MSG_628 : BOOL ;	//Leitungsschutzschalter Drehzahl Überwachung hat ausgelöst
   MSG_629 : BOOL ;	//Leitungsschutzschalter Netzteil Werkzeugwechsler hat ausgelöst
   MSG_630 : BOOL ;	//Leitungsschutzschalter Werkzeugidentifikation hat ausgelöst
   MSG_631 : BOOL ;	//Leitungsschutzschalter Werkzeugkegelreinigung hat ausgelöst
   MSG_632 : BOOL ;	//Leitungsschutzschalter Steuerstromkreis Palettenspeiche/-wechsler hat ausgelöst
   MSG_633 : BOOL ;	//Leitungsschutzschalter Bremse Palettenspeicher/-wechsler hat ausgelöst
   MSG_634 : BOOL ;	//Leitungsschutzschalter Betriebsdatenerfassung hat ausgelöst
   MSG_635 : BOOL ;	//Leitungsschutzschalter Werkzeugbruchüberwachung hat ausgelöst
   MSG_636 : BOOL ;	//Leitungsschutzschalter Minimalmengenschmierung hat ausgelöst
   MSG_637 : BOOL ;	//Leitungsschutzschalter Tuning IM 151_4 hat ausgelöst
   MSG_638 : BOOL ;	//Leitungsschutzschalter Tuning Ausgänge IM 151 hat ausgelöst
   MSG_639 : BOOL ;	//Leitungsschutzschalter Tuning Eingänge IM 151 hat ausgelöst
   MSG_640 : BOOL ;	//Leitungsschutzschalter Schaltschrankbeleuchtung hat ausgelöst
   MSG_641 : BOOL ;	//Leitungsschutzschalter Tuning IM 151_7 hat ausgelöst
   MSG_642 : BOOL ;	//Leitungsschutzschalter Drehzahl Überwachung Rüstplatz hat ausgelöst
   MSG_643 : BOOL ;	//Leitungsschutzschalter Messtaster hat ausgelöst
   MSG_644 : BOOL ;	//Leitungsschutzschalter Kabinentüre hat ausgelöst
   MSG_645 : BOOL ;	//Leitungsschutzschalter Leistung Spindel hat ausgelöst
   MSG_646 : BOOL ;	//Leitungsschutzschalter 230V hat ausgelöst
   MSG_647 : BOOL ;	//Leitungsschutzschalter 24V hat ausgelöst
   Me648 : BOOL ;	//1-
   Me649 : BOOL ;	//1-
   MSG_650 : BOOL ;	//TMS: Leitungsschutzschalter Bremse hat ausgelöst
   MSG_651 : BOOL ;	//TMS: Leitungsschutzschalter AC-Steuerspannung hat ausgelöst
   MSG_652 : BOOL ;	//TMS: Leitungsschutzschalter Steuerstromkreis hat ausgelöst
   MSG_653 : BOOL ;	//TMS: Leitungsschutzschalter Werkzeugeingabestation hat ausgelöst
   MSG_654 : BOOL ;	//TMS: Leitungsschutzschalter Ausgänge hat ausgelöst
   MSG_655 : BOOL ;	//TMS: Leitungsschutzschalter Netzteil hat ausgelöst
   Me656 : BOOL ;	//1-
   Me657 : BOOL ;	//1-
   MSG_658 : BOOL ;	//KSA: Leitungsschutzschalter Sensoren hat ausgelöst
   MSG_659 : BOOL ;	//KSA: Leitungsschutzschalter Proportionalventil 1 hat ausgelöst
   MSG_660 : BOOL ;	//KSA: Leitungsschutzschalter Proportionalventil 2 hat ausgelöst
   Me661 : BOOL ;	//1-
   Me662 : BOOL ;	//1-
   Me663 : BOOL ;	//1-
   Me664 : BOOL ;	//1-
   Me665 : BOOL ;	//1-
   Me666 : BOOL ;	//1-
   Me667 : BOOL ;	//1-
   Me668 : BOOL ;	//1-
   Me669 : BOOL ;	//1-
   Me670 : BOOL ;	//1-
   Me671 : BOOL ;	//1-
   Me672 : BOOL ;	//1-
   Me673 : BOOL ;	//1-
   Me674 : BOOL ;	//1-
   Me675 : BOOL ;	//1-
   MSG_676 : BOOL ;	//Leistungsschalter Späneförderer 2 hat ausgelöst
   MSG_677 : BOOL ;	//Leistungsschalter Kabinentüre hat ausgelöst
   MSG_678 : BOOL ;	//Leistungsschalter Steckdose Bedienpult hat ausgelöst
   MSG_679 : BOOL ;	//Leistungsschalter Steckdose Palettenwechsler hat ausgelöst
   MSG_680 : BOOL ;	//Leistungsschalter Schaltschrankbeleuchtung hat ausgelöst
   MSG_681 : BOOL ;	//Leistungsschalter DC-Steuerspannung_1 hat ausgelöst
   MSG_682 : BOOL ;	//Leistungsschalter DC-Steuerspannung_2 hat ausgelöst
   MSG_683 : BOOL ;	//Leistungsschalter AC-Steurspannung hat ausgelöst
   MSG_684 : BOOL ;	//Leistungsschalter Kühl-/Heizaggregat hat ausgelöst
   MSG_685 : BOOL ;	//Leistungsschalter AC-Versorgungsmodul hat ausgelöst
   MSG_686 : BOOL ;	//Leistungsschalter Lüfter AC hat ausgelöst
   MSG_687 : BOOL ;	//Leistungsschalter Kühlaggregat Schaltschrank hat ausgelöst
   MSG_688 : BOOL ;	//Leistungsschalter Werkzeugregal hat ausgelöst
   MSG_689 : BOOL ;	//Leistungsschalter Lüfter FD hat ausgelöst
   MSG_690 : BOOL ;	//Leistungsschalter Kühlmittelanlage hat ausgelöst
   Me691 : BOOL ;	//1-
   Me692 : BOOL ;	//1-
   MSG_693 : BOOL ;	//TMS: Leistungsschalter AC-Steuerspannung hat ausgelöst
   MSG_694 : BOOL ;	//TMS: Leistungsschalter Antriebe hat ausgelöst
   Me695 : BOOL ;	//1-
   Me696 : BOOL ;	//1-
   Me697 : BOOL ;	//1-
   Me698 : BOOL ;	//1-
   Me699 : BOOL ;	//1-
   MSG_700 : BOOL ;	//KSA: Leistungsschalter Pumpe Spänespülung Dach hat ausgelöst
   MSG_701 : BOOL ;	//KSA: Leistungsschalter Pumpe Spülpistole hat ausgelöst
   MSG_702 : BOOL ;	//KSA: Leistungsschalter Pumpe Spänespülung Türe hat ausgelöst
   MSG_703 : BOOL ;	//KSA: Leistungsschalter Pumpe Feinstbereich hat ausgelöst
   MSG_704 : BOOL ;	//KSA: Leistungsschalter Kratzerförder hat ausgelöst
   MSG_705 : BOOL ;	//KSA: Leistungsschalter Pumpe Kühlmittel 1 hat ausgelöst
   MSG_706 : BOOL ;	//KSA: Hauptschalter Kühlmittelanlage hat ausgelöst
   MSG_707 : BOOL ;	//KSA: Leistungsschalter Pumpe 40b hat ausgelöst
   MSG_708 : BOOL ;	//KSA: Leistungsschalter Pumpe 80b hat ausgelöst
   Me709 : BOOL ;	//1-
   Me710 : BOOL ;	//1-
   Me711 : BOOL ;	//1-
   Me712 : BOOL ;	//1-
   Me713 : BOOL ;	//1-
   Me714 : BOOL ;	//1-
   MSG_715 : BOOL ;	//KSA-Temp: Leistungsschalter Kompressor hat ausgelöst
   MSG_716 : BOOL ;	//KSA-Temp: Leistungsschalter Lüfter hat ausgelöst
   MSG_717 : BOOL ;	//KSA-Temp: Leistungsschalter Rührwerk hat ausgelöst
   MSG_718 : BOOL ;	//KSA-Temp: Leistungsschalter Hebepumpe hat ausgelöst
   MSG_719 : BOOL ;	//KSA-Temp: Leistungsschalter Heizung hat ausgelöst
   MSG_720 : BOOL ;	//KSA-Temp: Leistungsschalter Steuerspannung hat ausgelöst
   Me721 : BOOL ;	//1-
   Me722 : BOOL ;	//1-
   Me723 : BOOL ;	//1-
   Me724 : BOOL ;	//1-
   MSG_725 : BOOL ;	//Wartungstüre Werkzeugmagazin ist offen
   MSG_726 : BOOL ;	//Wartungstüre Werkzeugregal ist offen
   MSG_727 : BOOL ;	//Wartungstüre Werkzeugeingabestation ist offen
   MSG_728 : BOOL ;	//Wartungstüre Palettenspeicher/-wechsler ist offen
   Me729 : BOOL ;	//1-
   Me730 : BOOL ;	//1-
   Me731 : BOOL ;	//1-
   Me732 : BOOL ;	//1-
   Me733 : BOOL ;	//1-
   Me734 : BOOL ;	//1-
   Me735 : BOOL ;	//1-
   Me736 : BOOL ;	//1-
   MSG_737 : BOOL ;	//Zeitüberschreitung beim Öffnen der linken Rüstplatztür
   MSG_738 : BOOL ;	//Zeitüberschreitung beim Schließen der linken Rüstplatztür
   MSG_739 : BOOL ;	//Zeitüberschreitung beim Öffnen der rechten Rüstplatztür
   MSG_740 : BOOL ;	//Zeitüberschreitung beim Schließen der rechten Rüstplatztür
   MSG_741 : BOOL ;	//Öffnen der Rüstplatztüre(n) nicht möglich
   MSG_742 : BOOL ;	//Manuelle Bedienung der Rüstplatztüre(n) nicht möglich
   MSG_743 : BOOL ;	//Warte mit Palettenfreigabe bis Rüstplatztüre(n) verriegelt
   MSG_744 : BOOL ;	//Steuerung der Rüstplatztüre(n) - ungültiger Betriebsmodus!
   Me745 : BOOL ;	//1-
   Me746 : BOOL ;	//1-
   Me747 : BOOL ;	//1-
   Me748 : BOOL ;	//1-
   Me749 : BOOL ;	//1-
   Me750 : BOOL ;	//1-
   Me751 : BOOL ;	//1-
   Me752 : BOOL ;	//1-
   Me753 : BOOL ;	//1-
   Me754 : BOOL ;	//1-
   Me755 : BOOL ;	//1-
   Me756 : BOOL ;	//1-
   Me757 : BOOL ;	//1-
   Me758 : BOOL ;	//1-
   Me759 : BOOL ;	//1-
   Me760 : BOOL ;	//1-
   Me761 : BOOL ;	//1-
   Me762 : BOOL ;	//1-
   Me763 : BOOL ;	//1-
   Me764 : BOOL ;	//1-
   Me765 : BOOL ;	//1-
   Me766 : BOOL ;	//1-
   Me767 : BOOL ;	//1-
   Me768 : BOOL ;	//1-
   Me769 : BOOL ;	//1-
   Me770 : BOOL ;	//1-
   Me771 : BOOL ;	//1-
   Me772 : BOOL ;	//1-
   Me773 : BOOL ;	//1-
   Me774 : BOOL ;	//1-
   Me775 : BOOL ;	//1-
   Me776 : BOOL ;	//1-
   Me777 : BOOL ;	//1-
   Me778 : BOOL ;	//1-
   Me779 : BOOL ;	//1-
   Me780 : BOOL ;	//1-
   Me781 : BOOL ;	//1-
   Me782 : BOOL ;	//1-
   Me783 : BOOL ;	//1-
   Me784 : BOOL ;	//1-
   Me785 : BOOL ;	//1-
   Me786 : BOOL ;	//1-
   Me787 : BOOL ;	//1-
   Me788 : BOOL ;	//1-
   Me789 : BOOL ;	//1-
   Me790 : BOOL ;	//1-
   Me791 : BOOL ;	//1-
   Me792 : BOOL ;	//1-
   Me793 : BOOL ;	//1-
   Me794 : BOOL ;	//1-
   Me795 : BOOL ;	//1-
   Me796 : BOOL ;	//1-
   Me797 : BOOL ;	//1-
   Me798 : BOOL ;	//1-
   Me799 : BOOL ;	//1-
   MSG_800 : BOOL ;	//LUB: Druck an Schmierverteiler NC-Rundtisch nicht erreicht
   MSG_801 : BOOL ;	//LUB: Zeitüberschreitung beim Abschalten der Schmierung (NC-Rundtisch)
   Me802 : BOOL ;	//1-
   Me803 : BOOL ;	//1-
   Me804 : BOOL ;	//1-
   Me805 : BOOL ;	//1-
   Me806 : BOOL ;	//1-
   Me807 : BOOL ;	//1-
   Me808 : BOOL ;	//1-
   Me809 : BOOL ;	//1-
   Me810 : BOOL ;	//1-
   Me811 : BOOL ;	//1-
   Me812 : BOOL ;	//1-
   Me813 : BOOL ;	//1-
   Me814 : BOOL ;	//1-
   Me815 : BOOL ;	//1-
   Me816 : BOOL ;	//1-
   Me817 : BOOL ;	//1-
   Me818 : BOOL ;	//1-
   Me819 : BOOL ;	//1-
   Me820 : BOOL ;	//1-
   Me821 : BOOL ;	//1-
   Me822 : BOOL ;	//1-
   Me823 : BOOL ;	//1-
   Me824 : BOOL ;	//1-
   Me825 : BOOL ;	//1-
   Me826 : BOOL ;	//1-
   Me827 : BOOL ;	//1-
   Me828 : BOOL ;	//1-
   Me829 : BOOL ;	//1-
   Me830 : BOOL ;	//1-
   Me831 : BOOL ;	//1-
   Me832 : BOOL ;	//1-
   Me833 : BOOL ;	//1-
   Me834 : BOOL ;	//1-
   Me835 : BOOL ;	//1-
   Me836 : BOOL ;	//1-
   Me837 : BOOL ;	//1-
   Me838 : BOOL ;	//1-
   Me839 : BOOL ;	//1-
   Me840 : BOOL ;	//1-
   Me841 : BOOL ;	//1-
   Me842 : BOOL ;	//1-
   Me843 : BOOL ;	//1-
   Me844 : BOOL ;	//1-
   Me845 : BOOL ;	//1-
   Me846 : BOOL ;	//1-
   Me847 : BOOL ;	//1-
   Me848 : BOOL ;	//1-
   Me849 : BOOL ;	//1-
   Me850 : BOOL ;	//1-
   Me851 : BOOL ;	//1-
   Me852 : BOOL ;	//1-
   Me853 : BOOL ;	//1-
   Me854 : BOOL ;	//1-
   Me855 : BOOL ;	//1-
   Me856 : BOOL ;	//1-
   Me857 : BOOL ;	//1-
   Me858 : BOOL ;	//1-
   Me859 : BOOL ;	//1-
   Me860 : BOOL ;	//1-
   Me861 : BOOL ;	//1-
   Me862 : BOOL ;	//1-
   Me863 : BOOL ;	//1-
   Me864 : BOOL ;	//1-
   Me865 : BOOL ;	//1-
   Me866 : BOOL ;	//1-
   Me867 : BOOL ;	//1-
   Me868 : BOOL ;	//1-
   Me869 : BOOL ;	//1-
   Me870 : BOOL ;	//1-
   Me871 : BOOL ;	//1-
   Me872 : BOOL ;	//1-
   Me873 : BOOL ;	//1-
   Me874 : BOOL ;	//1-
   Me875 : BOOL ;	//1-
   Me876 : BOOL ;	//1-
   Me877 : BOOL ;	//1-
   Me878 : BOOL ;	//1-
   Me879 : BOOL ;	//1-
   Me880 : BOOL ;	//1-
   Me881 : BOOL ;	//1-
   Me882 : BOOL ;	//1-
   Me883 : BOOL ;	//1-
   Me884 : BOOL ;	//1-
   Me885 : BOOL ;	//1-
   Me886 : BOOL ;	//1-
   Me887 : BOOL ;	//1-
   Me888 : BOOL ;	//1-
   Me889 : BOOL ;	//1-
   Me890 : BOOL ;	//1-
   Me891 : BOOL ;	//1-
   Me892 : BOOL ;	//1-
   Me893 : BOOL ;	//1-
   Me894 : BOOL ;	//1-
   Me895 : BOOL ;	//1-
   Me896 : BOOL ;	//1-
   Me897 : BOOL ;	//1-
   Me898 : BOOL ;	//1-
   Me899 : BOOL ;	//1-
   Me900 : BOOL ;	//1-
   Me901 : BOOL ;	//1-
   Me902 : BOOL ;	//1-
   Me903 : BOOL ;	//1-
   Me904 : BOOL ;	//1-
   Me905 : BOOL ;	//1-
   Me906 : BOOL ;	//1-
   Me907 : BOOL ;	//1-
   Me908 : BOOL ;	//1-
   Me909 : BOOL ;	//1-
   Me910 : BOOL ;	//1-
   Me911 : BOOL ;	//1-
   Me912 : BOOL ;	//1-
   Me913 : BOOL ;	//1-
   Me914 : BOOL ;	//1-
   Me915 : BOOL ;	//1-
   Me916 : BOOL ;	//1-
   Me917 : BOOL ;	//1-
   Me918 : BOOL ;	//1-
   Me919 : BOOL ;	//1-
   Me920 : BOOL ;	//1-
   Me921 : BOOL ;	//1-
   Me922 : BOOL ;	//1-
   Me923 : BOOL ;	//1-
   Me924 : BOOL ;	//1-
   Me925 : BOOL ;	//1-
   Me926 : BOOL ;	//1-
   Me927 : BOOL ;	//1-
   Me928 : BOOL ;	//1-
   Me929 : BOOL ;	//1-
   Me930 : BOOL ;	//1-
   Me931 : BOOL ;	//1-
   Me932 : BOOL ;	//1-
   Me933 : BOOL ;	//1-
   Me934 : BOOL ;	//1-
   Me935 : BOOL ;	//1-
   Me936 : BOOL ;	//1-
   Me937 : BOOL ;	//1-
   Me938 : BOOL ;	//1-
   Me939 : BOOL ;	//1-
   Me940 : BOOL ;	//1-
   Me941 : BOOL ;	//1-
   Me942 : BOOL ;	//1-
   Me943 : BOOL ;	//1-
   Me944 : BOOL ;	//1-
   Me945 : BOOL ;	//1-
   Me946 : BOOL ;	//1-
   Me947 : BOOL ;	//1-
   Me948 : BOOL ;	//1-
   Me949 : BOOL ;	//1-
   Me950 : BOOL ;	//1-
   Me951 : BOOL ;	//1-
   Me952 : BOOL ;	//1-
   Me953 : BOOL ;	//1-
   Me954 : BOOL ;	//1-
   Me955 : BOOL ;	//1-
   Me956 : BOOL ;	//1-
   Me957 : BOOL ;	//1-
   Me958 : BOOL ;	//1-
   Me959 : BOOL ;	//1-
   Me960 : BOOL ;	//1-
   Me961 : BOOL ;	//1-
   Me962 : BOOL ;	//1-
   Me963 : BOOL ;	//1-
   Me964 : BOOL ;	//1-
   Me965 : BOOL ;	//1-
   Me966 : BOOL ;	//1-
   Me967 : BOOL ;	//1-
   Me968 : BOOL ;	//1-
   Me969 : BOOL ;	//1-
   Me970 : BOOL ;	//1-
   Me971 : BOOL ;	//1-
   Me972 : BOOL ;	//1-
   Me973 : BOOL ;	//1-
   Me974 : BOOL ;	//1-
   Me975 : BOOL ;	//1-
   Me976 : BOOL ;	//1-
   Me977 : BOOL ;	//1-
   Me978 : BOOL ;	//1-
   Me979 : BOOL ;	//1-
   Me980 : BOOL ;	//1-
   Me981 : BOOL ;	//1-
   Me982 : BOOL ;	//1-
   Me983 : BOOL ;	//1-
   Me984 : BOOL ;	//1-
   Me985 : BOOL ;	//1-
   Me986 : BOOL ;	//1-
   Me987 : BOOL ;	//1-
   Me988 : BOOL ;	//1-
   Me989 : BOOL ;	//1-
   Me990 : BOOL ;	//1-
   Me991 : BOOL ;	//1-
   Me992 : BOOL ;	//1-
   Me993 : BOOL ;	//1-
   Me994 : BOOL ;	//1-
   Me995 : BOOL ;	//1-
   Me996 : BOOL ;	//1-
   Me997 : BOOL ;	//1-
   Me998 : BOOL ;	//1-
   Me999 : BOOL ;	//1-
   Me1000 : BOOL ;	//1-
   Me1001 : BOOL ;	//1-
   Me1002 : BOOL ;	//1-
   Me1003 : BOOL ;	//1-
   Me1004 : BOOL ;	//1-
   Me1005 : BOOL ;	//1-
   Me1006 : BOOL ;	//1-
   Me1007 : BOOL ;	//1-
   Me1008 : BOOL ;	//1-
   Me1009 : BOOL ;	//1-
   Me1010 : BOOL ;	//1-
   Me1011 : BOOL ;	//1-
   Me1012 : BOOL ;	//1-
   Me1013 : BOOL ;	//1-
   Me1014 : BOOL ;	//1-
   Me1015 : BOOL ;	//1-
   Me1016 : BOOL ;	//1-
   Me1017 : BOOL ;	//1-
   Me1018 : BOOL ;	//1-
   Me1019 : BOOL ;	//1-
   Me1020 : BOOL ;	//1-
   Me1021 : BOOL ;	//1-
   Me1022 : BOOL ;	//1-
   Me1023 : BOOL ;	//1-
   Me1024 : BOOL ;	//1-
  END_STRUCT ;	
END_TYPE

TYPE "UDT101"	// UDT 101
AUTHOR : SPAC_slh
VERSION : 0.1
  STRUCT
   T : ARRAY  [0 .. 31 ] OF UDT 1010;
  END_STRUCT ;	
END_TYPE

TYPE "UDT1010"	// UDT 1010
AUTHOR : SPAC_slh
VERSION : 0.1
  STRUCT
   SwT : ARRAY  [0 .. 2 ] OF //SwZeit[0]
   TIME ;
   x : STRUCT
    E1gs : BOOL ;	//Endlage 1 gespeichert
    E2gs : BOOL ;	//Endlage 2 gespeichert
    x2 : BOOL ;
    x3 : BOOL ;
    x4 : BOOL ;
    x5 : BOOL ;
    x6 : BOOL ;
    x7 : BOOL ;
    fk0 : BOOL ;
    fk1 : BOOL ;
    fk2 : BOOL ;
    fk3 : BOOL ;
    fk4 : BOOL ;
    fk5 : BOOL ;
    fk6 : BOOL ;
    fk7 : BOOL ;
   END_STRUCT ;
  END_STRUCT ;	
END_TYPE

